// TwinCAT 3 PLC project SiasunDemo
// Title: ServoDriveDemo
// Company: Siasun
// ProjectVersion: 0.1.0
// ProgramVersion: 3.1.0.9
// libraries:
//   Tc2_EtherCAT, * (Beckhoff Automation GmbH)
//   Tc2_MC2, * (Beckhoff Automation GmbH)
//   Tc2_Standard, * (Beckhoff Automation GmbH)
//   Tc2_System, * (Beckhoff Automation GmbH)
//   Tc2_Utilities, * (Beckhoff Automation GmbH)
//   Tc2_XmlDataSrv, * (Beckhoff Automation GmbH)
//   Tc3_JsonXml, * (Beckhoff Automation GmbH)
//   Tc3_Module, * (Beckhoff Automation GmbH)
//   VisuDialogs, * (System)
// project tree:
//   DUTs/ Para.TcDUT, Struct_AxisDrive.TcDUT (not stored), Struct_AxisXmlRW.TcDUT, Struct_EndDrive.TcDUT, Struct_MotionPara.TcDUT, Struct_PLCVersion.TcDUT (not stored), Struct_AxisInfo.TcDUT (not stored), Struct_AxisStatus.TcDUT (not stored), Struct_ServoAccessParameters.TcDUT (not stored), Struct_ObservedParameters.TcDUT
//   / GlobalTextList.TcGTLO, PlcTask.TcTTO (not stored), 视图管理器.TcVMO (not stored)
//   POUs/CoeSdoRW/ AmsNetID_TO_TAmsNetID.TcPOU (not stored), FB_SDO_READ.TcPOU (not stored), FB_SDO_WRITE.TcPOU (not stored)
//   POUs/ FB_AxisOperate.TcPOU, MAIN.TcPOU (not stored)
//   VISUs/ StatJoint.TcVIS (not stored), StatJoint_6Axis.TcVIS
// real-time tasks:
//   TASK PlcTask: cycle T#4ms, priority 20, ADS port 350
//   TASK VISU_TASK: cycle T#200000us, priority 30, ADS port 351
//   TASK PlcTask1: cycle T#1ms, priority 21, ADS port 352
// motion (NC):
//   TASK NC-Task 1 SAF: cycle T#4ms, priority 4, ADS port 501
//   TASK NC-Task 1 SVB: cycle T#4ms, priority 8, ADS port 511
//   AXIS Axis 1 (id 1)
//     PositionAreaControl: Enable=false
//     TargetPosControl: Enable=false
//     OtherSettings: AllowMotionCmdToSlave=true
//     encoder EncType=19
//       EncPara: ScaleFactorNumerator=0.000686645507813, EncMode=3, MaxCount=#xffffffff, ReferenceSystem=1
//         Inc: RefSyncInverse=false
//     drive DrvType=16
//       DrvPara: MaxCount=#xffffffff, DriveControlDWord=#x00020000
//         Analog: TorqueSetpointScale=10
//         TimeComp: TaskDelayCycles=1
//     controller CtrType=1
//       CtrPara: PriorControlFactor=1
//         PosDiffControl: Enable=false
//         Observer: BandWidth=20
//   AXIS Axis 2 (id 2)
//     PositionAreaControl: Enable=false
//     TargetPosControl: Enable=false
//     OtherSettings: AllowMotionCmdToSlave=true
//     encoder EncType=19
//       EncPara: ScaleFactorNumerator=0.000686645507813, EncMode=3, MaxCount=#xffffffff, ReferenceSystem=1
//         Inc: RefSyncInverse=false
//     drive DrvType=16
//       DrvPara: MaxCount=#xffffffff, DriveControlDWord=#x00020000
//         Analog: TorqueSetpointScale=10
//         TimeComp: TaskDelayCycles=1
//     controller CtrType=1
//       CtrPara: PriorControlFactor=1
//         PosDiffControl: Enable=false
//         Observer: BandWidth=20
//   AXIS Axis 3 (id 3)
//     PositionAreaControl: Enable=false
//     TargetPosControl: Enable=false
//     OtherSettings: AllowMotionCmdToSlave=true
//     encoder EncType=19
//       EncPara: ScaleFactorNumerator=0.000686645507813, EncMode=3, MaxCount=#xffffffff, ReferenceSystem=1
//         Inc: RefSyncInverse=false
//     drive DrvType=16
//       DrvPara: MaxCount=#xffffffff, DriveControlDWord=#x00020000
//         TimeComp: TaskDelayCycles=1
//     controller CtrType=1
//       CtrPara: PriorControlFactor=1
//         PosDiffControl: Enable=false
//         Observer: BandWidth=20
//   AXIS Axis 4 (id 4)
//     PositionAreaControl: Enable=false
//     TargetPosControl: Enable=false
//     OtherSettings: AllowMotionCmdToSlave=true
//     encoder EncType=19
//       EncPara: ScaleFactorNumerator=0.000686645507813, EncMode=3, MaxCount=#xffffffff, ReferenceSystem=1
//         Inc: RefSyncInverse=false
//     drive DrvType=16
//       DrvPara: MaxCount=#xffffffff, DriveControlDWord=#x00020000
//         TimeComp: TaskDelayCycles=1
//     controller CtrType=1
//       CtrPara: PriorControlFactor=1
//         PosDiffControl: Enable=false
//         Observer: BandWidth=20
//   AXIS Axis 5 (id 5)
//     PositionAreaControl: Enable=false
//     TargetPosControl: Enable=false
//     OtherSettings: AllowMotionCmdToSlave=true
//     encoder EncType=19
//       EncPara: ScaleFactorNumerator=0.000686645507813, EncMode=3, MaxCount=#xffffffff, ReferenceSystem=1
//         Inc: RefSyncInverse=false
//     drive DrvType=16
//       DrvPara: MaxCount=#xffffffff, DriveControlDWord=#x00020000
//         TimeComp: TaskDelayCycles=1
//     controller CtrType=1
//       CtrPara: PriorControlFactor=1
//         PosDiffControl: Enable=false
//         Observer: BandWidth=20
//   AXIS Axis 6 (id 6)
//     PositionAreaControl: Enable=false
//     TargetPosControl: Enable=false
//     OtherSettings: AllowMotionCmdToSlave=true
//     encoder EncType=19
//       EncPara: ScaleFactorNumerator=0.000686645507813, EncMode=3, MaxCount=#xffffffff, ReferenceSystem=1
//         Inc: RefSyncInverse=false
//     drive DrvType=16
//       DrvPara: MaxCount=#xffffffff, DriveControlDWord=#x00020000
//         TimeComp: TaskDelayCycles=1
//     controller CtrType=1
//       CtrPara: PriorControlFactor=1
//         PosDiffControl: Enable=false
//         Observer: BandWidth=20
//   AXIS Axis 7 (id 7)
//     PositionAreaControl: Enable=false
//     TargetPosControl: Enable=false
//     OtherSettings: AllowMotionCmdToSlave=true
//     encoder EncType=19
//       EncPara: ScaleFactorNumerator=0.000686645507813, MaxCount=#xffffffff
//         Inc: RefSyncInverse=false
//     drive DrvType=16
//       DrvPara: MaxCount=#xffffffff
//         TimeComp: TaskDelayCycles=1
//     controller CtrType=1
//       CtrPara: PriorControlFactor=1
//         PosDiffControl: Enable=false
//         Observer: BandWidth=20
// I/O:
//   DEVICE Device 3 (EtherCAT), AmsNetId 172.16.3.61.4.1
//     Term 8 (EK1200) [EK1200-5000 EtherCAT Power supply (2A E-Bus)]
//       Term 8 (EK1110) [EK1110 EtherCAT extension]
//     Drive 9 (SERVO_ECAT) [SERVO_ECAT]
//     Drive 10 (SERVO_ECAT) [SERVO_ECAT]
//     Drive 11 (SERVO_ECAT) [SERVO_ECAT] (disabled)
//     Drive 12 (SERVO_ECAT) [SERVO_ECAT]
//     Drive 13 (SERVO_ECAT) [SERVO_ECAT]
//     Drive 14 (SERVO_ECAT) [SERVO_ECAT]
//     Box 15 (ECAT_EndIO) [ECAT_EndIO]
// variable links:
//   NC-Task 1 SAF/Axes/Axis 1 <-> Device 3 (EtherCAT)/Drive 9 (SERVO_ECAT)
//     Drive/Inputs/In/nDataIn3[0] <-> Input mapping 0/TorqueActualValue1
//     Drive/Inputs/In/nState1 <-> Input mapping 0/StatusWord
//     Drive/Inputs/In/nState2 <-> Input mapping 0/StatusWord @bit 8
//     Drive/Inputs/In/nState4 @bit 1 <-> WcState/InputToggle
//     Drive/Inputs/In/nState4 <-> WcState/WcState
//     Drive/Inputs/In/nState5 <-> Input mapping 0/ModesOfOperationDisplay
//     Drive/Outputs/Out/nCtrl1 <-> Output mapping 0/ControlWord
//     Drive/Outputs/Out/nCtrl2 <-> Output mapping 0/ControlWord @bit 8
//     Drive/Outputs/Out/nDataOut1 <-> Output mapping 0/TargetPosition
//     Enc/Inputs/In/nDataIn1 <-> Input mapping 0/PositionActualValue
//     Enc/Inputs/In/nState4 @bit 1 <-> WcState/InputToggle
//     Enc/Inputs/In/nState4 <-> WcState/WcState
//   NC-Task 1 SAF/Axes/Axis 2 <-> Device 3 (EtherCAT)/Drive 10 (SERVO_ECAT)
//     Drive/Inputs/In/nDataIn3[0] <-> Input mapping 0/TorqueActualValue1
//     Drive/Inputs/In/nState1 <-> Input mapping 0/StatusWord
//     Drive/Inputs/In/nState2 <-> Input mapping 0/StatusWord @bit 8
//     Drive/Inputs/In/nState4 @bit 1 <-> WcState/InputToggle
//     Drive/Inputs/In/nState4 <-> WcState/WcState
//     Drive/Inputs/In/nState5 <-> Input mapping 0/ModesOfOperationDisplay
//     Drive/Outputs/Out/nCtrl1 <-> Output mapping 0/ControlWord
//     Drive/Outputs/Out/nCtrl2 <-> Output mapping 0/ControlWord @bit 8
//     Drive/Outputs/Out/nDataOut1 <-> Output mapping 0/TargetPosition
//     Enc/Inputs/In/nDataIn1 <-> Input mapping 0/PositionActualValue
//     Enc/Inputs/In/nState4 @bit 1 <-> WcState/InputToggle
//     Enc/Inputs/In/nState4 <-> WcState/WcState
//   NC-Task 1 SAF/Axes/Axis 3 <-> Device 3 (EtherCAT)/Drive 11 (SERVO_ECAT)
//     Drive/Inputs/In/nDataIn3[0] <-> Input mapping 0/TorqueActualValue1
//     Drive/Inputs/In/nState1 <-> Input mapping 0/StatusWord
//     Drive/Inputs/In/nState2 <-> Input mapping 0/StatusWord @bit 8
//     Drive/Inputs/In/nState4 @bit 1 <-> WcState/InputToggle
//     Drive/Inputs/In/nState4 <-> WcState/WcState
//     Drive/Inputs/In/nState5 <-> Input mapping 0/ModesOfOperationDisplay
//     Drive/Outputs/Out/nCtrl1 <-> Output mapping 0/ControlWord
//     Drive/Outputs/Out/nCtrl2 <-> Output mapping 0/ControlWord @bit 8
//     Drive/Outputs/Out/nDataOut1 <-> Output mapping 0/TargetPosition
//     Enc/Inputs/In/nDataIn1 <-> Input mapping 0/PositionActualValue
//     Enc/Inputs/In/nState4 @bit 1 <-> WcState/InputToggle
//     Enc/Inputs/In/nState4 <-> WcState/WcState
//   NC-Task 1 SAF/Axes/Axis 4 <-> Device 3 (EtherCAT)/Drive 12 (SERVO_ECAT)
//     Drive/Inputs/In/nDataIn3[0] <-> Input mapping 0/TorqueActualValue1
//     Drive/Inputs/In/nState1 <-> Input mapping 0/StatusWord
//     Drive/Inputs/In/nState2 <-> Input mapping 0/StatusWord @bit 8
//     Drive/Inputs/In/nState4 @bit 1 <-> WcState/InputToggle
//     Drive/Inputs/In/nState4 <-> WcState/WcState
//     Drive/Inputs/In/nState5 <-> Input mapping 0/ModesOfOperationDisplay
//     Drive/Outputs/Out/nCtrl1 <-> Output mapping 0/ControlWord
//     Drive/Outputs/Out/nCtrl2 <-> Output mapping 0/ControlWord @bit 8
//     Drive/Outputs/Out/nDataOut1 <-> Output mapping 0/TargetPosition
//     Enc/Inputs/In/nDataIn1 <-> Input mapping 0/PositionActualValue
//     Enc/Inputs/In/nState4 @bit 1 <-> WcState/InputToggle
//     Enc/Inputs/In/nState4 <-> WcState/WcState
//   NC-Task 1 SAF/Axes/Axis 5 <-> Device 3 (EtherCAT)/Drive 13 (SERVO_ECAT)
//     Drive/Inputs/In/nDataIn3[0] <-> Input mapping 0/TorqueActualValue1
//     Drive/Inputs/In/nState1 <-> Input mapping 0/StatusWord
//     Drive/Inputs/In/nState2 <-> Input mapping 0/StatusWord @bit 8
//     Drive/Inputs/In/nState4 @bit 1 <-> WcState/InputToggle
//     Drive/Inputs/In/nState4 <-> WcState/WcState
//     Drive/Inputs/In/nState5 <-> Input mapping 0/ModesOfOperationDisplay
//     Drive/Outputs/Out/nCtrl1 <-> Output mapping 0/ControlWord
//     Drive/Outputs/Out/nCtrl2 <-> Output mapping 0/ControlWord @bit 8
//     Drive/Outputs/Out/nDataOut1 <-> Output mapping 0/TargetPosition
//     Enc/Inputs/In/nDataIn1 <-> Input mapping 0/PositionActualValue
//     Enc/Inputs/In/nState4 @bit 1 <-> WcState/InputToggle
//     Enc/Inputs/In/nState4 <-> WcState/WcState
//   NC-Task 1 SAF/Axes/Axis 6 <-> Device 3 (EtherCAT)/Drive 14 (SERVO_ECAT)
//     Drive/Inputs/In/nDataIn3[0] <-> Input mapping 0/TorqueActualValue1
//     Drive/Inputs/In/nState1 <-> Input mapping 0/StatusWord
//     Drive/Inputs/In/nState2 <-> Input mapping 0/StatusWord @bit 8
//     Drive/Inputs/In/nState4 @bit 1 <-> WcState/InputToggle
//     Drive/Inputs/In/nState4 <-> WcState/WcState
//     Drive/Inputs/In/nState5 <-> Input mapping 0/ModesOfOperationDisplay
//     Drive/Outputs/Out/nCtrl1 <-> Output mapping 0/ControlWord
//     Drive/Outputs/Out/nCtrl2 <-> Output mapping 0/ControlWord @bit 8
//     Drive/Outputs/Out/nDataOut1 <-> Output mapping 0/TargetPosition
//     Enc/Inputs/In/nDataIn1 <-> Input mapping 0/PositionActualValue
//     Enc/Inputs/In/nState4 @bit 1 <-> WcState/InputToggle
//     Enc/Inputs/In/nState4 <-> WcState/WcState
//   SiasunDemo/SiasunDemo Instance <-> Device 3 (EtherCAT)/Box 15 (ECAT_EndIO)
//     PlcTask Inputs/MAIN.EndInfo.EC_State <-> InfoData/State
//     PlcTask Inputs/MAIN.EndInfo.WC_State <-> WcState/WcState
//     PlcTask Inputs/MAIN.EndInfo.nSlaveAddr <-> InfoData/AdsAddr/port
//     PlcTask Inputs/MAIN.EndInfo.sNetID <-> InfoData/AdsAddr/netId
//   SiasunDemo/SiasunDemo Instance <-> Device 3 (EtherCAT)/Drive 10 (SERVO_ECAT)
//     PlcTask Inputs/MAIN.AxisOp[1].AxisDrive.InfoData_StateJoint <-> InfoData/State
//     PlcTask Inputs/MAIN.AxisOp[1].AxisDrive.Joint_PositionActual <-> Input mapping 0/AuxiliaryPositionActualValue
//     PlcTask Inputs/MAIN.AxisOp[1].AxisDrive.Joint_VelocityActual <-> Input mapping 0/AuxiliaryVelocityActualValue
//     PlcTask Inputs/MAIN.AxisOp[1].AxisDrive.MoveMode <-> Input mapping 0/ModesOfOperationDisplay
//     PlcTask Inputs/MAIN.AxisOp[1].AxisDrive.ServoErrId <-> Input mapping 0/ErrorCode
//     PlcTask Inputs/MAIN.AxisOp[1].AxisDrive.StatusWord <-> Input mapping 0/StatusWord
//     PlcTask Inputs/MAIN.AxisOp[1].AxisDrive.TorqueValue <-> Input mapping 0/CurrentActualvalue
//     PlcTask Inputs/MAIN.AxisOp[1].AxisDrive.WC_State <-> WcState/WcState
//     PlcTask Inputs/MAIN.AxisOp[1].AxisDrive.nSlaveAddr <-> InfoData/AdsAddr/port
//     PlcTask Inputs/MAIN.AxisOp[1].AxisDrive.sNetID <-> InfoData/AdsAddr/netId
//     PlcTask Outputs/MAIN.AxisOp[1].AxisDrive.TargetMode <-> Output mapping 0/ModesOfOperation
//     PlcTask Outputs/MAIN.AxisOp[1].AxisDrive.TargetTorque <-> Output mapping 0/TargetTorque
//     PlcTask Outputs/MAIN.AxisOp[1].AxisDrive.TargetVelocity <-> Output mapping 0/TargetVelocity
//   SiasunDemo/SiasunDemo Instance <-> Device 3 (EtherCAT)/Drive 11 (SERVO_ECAT)
//     PlcTask Inputs/MAIN.AxisOp[2].AxisDrive.InfoData_StateJoint <-> InfoData/State
//     PlcTask Inputs/MAIN.AxisOp[2].AxisDrive.Joint_PositionActual <-> Input mapping 0/AuxiliaryPositionActualValue
//     PlcTask Inputs/MAIN.AxisOp[2].AxisDrive.Joint_VelocityActual <-> Input mapping 0/AuxiliaryVelocityActualValue
//     PlcTask Inputs/MAIN.AxisOp[2].AxisDrive.MoveMode <-> Input mapping 0/ModesOfOperationDisplay
//     PlcTask Inputs/MAIN.AxisOp[2].AxisDrive.ServoErrId <-> Input mapping 0/ErrorCode
//     PlcTask Inputs/MAIN.AxisOp[2].AxisDrive.StatusWord <-> Input mapping 0/StatusWord
//     PlcTask Inputs/MAIN.AxisOp[2].AxisDrive.TorqueValue <-> Input mapping 0/CurrentActualvalue
//     PlcTask Inputs/MAIN.AxisOp[2].AxisDrive.WC_State <-> WcState/WcState
//     PlcTask Inputs/MAIN.AxisOp[2].AxisDrive.nSlaveAddr <-> InfoData/AdsAddr/port
//     PlcTask Inputs/MAIN.AxisOp[2].AxisDrive.sNetID <-> InfoData/AdsAddr/netId
//     PlcTask Outputs/MAIN.AxisOp[2].AxisDrive.TargetMode <-> Output mapping 0/ModesOfOperation
//     PlcTask Outputs/MAIN.AxisOp[2].AxisDrive.TargetTorque <-> Output mapping 0/TargetTorque
//     PlcTask Outputs/MAIN.AxisOp[2].AxisDrive.TargetVelocity <-> Output mapping 0/TargetVelocity
//   SiasunDemo/SiasunDemo Instance <-> Device 3 (EtherCAT)/Drive 12 (SERVO_ECAT)
//     PlcTask Inputs/MAIN.AxisOp[3].AxisDrive.InfoData_StateJoint <-> InfoData/State
//     PlcTask Inputs/MAIN.AxisOp[3].AxisDrive.Joint_PositionActual <-> Input mapping 0/AuxiliaryPositionActualValue
//     PlcTask Inputs/MAIN.AxisOp[3].AxisDrive.Joint_VelocityActual <-> Input mapping 0/AuxiliaryVelocityActualValue
//     PlcTask Inputs/MAIN.AxisOp[3].AxisDrive.MoveMode <-> Input mapping 0/ModesOfOperationDisplay
//     PlcTask Inputs/MAIN.AxisOp[3].AxisDrive.ServoErrId <-> Input mapping 0/ErrorCode
//     PlcTask Inputs/MAIN.AxisOp[3].AxisDrive.StatusWord <-> Input mapping 0/StatusWord
//     PlcTask Inputs/MAIN.AxisOp[3].AxisDrive.TorqueValue <-> Input mapping 0/CurrentActualvalue
//     PlcTask Inputs/MAIN.AxisOp[3].AxisDrive.WC_State <-> WcState/WcState
//     PlcTask Inputs/MAIN.AxisOp[3].AxisDrive.nSlaveAddr <-> InfoData/AdsAddr/port
//     PlcTask Inputs/MAIN.AxisOp[3].AxisDrive.sNetID <-> InfoData/AdsAddr/netId
//     PlcTask Outputs/MAIN.AxisOp[3].AxisDrive.TargetMode <-> Output mapping 0/ModesOfOperation
//     PlcTask Outputs/MAIN.AxisOp[3].AxisDrive.TargetTorque <-> Output mapping 0/TargetTorque
//     PlcTask Outputs/MAIN.AxisOp[3].AxisDrive.TargetVelocity <-> Output mapping 0/TargetVelocity
//   SiasunDemo/SiasunDemo Instance <-> Device 3 (EtherCAT)/Drive 13 (SERVO_ECAT)
//     PlcTask Inputs/MAIN.AxisOp[4].AxisDrive.InfoData_StateJoint <-> InfoData/State
//     PlcTask Inputs/MAIN.AxisOp[4].AxisDrive.Joint_PositionActual <-> Input mapping 0/AuxiliaryPositionActualValue
//     PlcTask Inputs/MAIN.AxisOp[4].AxisDrive.Joint_VelocityActual <-> Input mapping 0/AuxiliaryVelocityActualValue
//     PlcTask Inputs/MAIN.AxisOp[4].AxisDrive.MoveMode <-> Input mapping 0/ModesOfOperationDisplay
//     PlcTask Inputs/MAIN.AxisOp[4].AxisDrive.ServoErrId <-> Input mapping 0/ErrorCode
//     PlcTask Inputs/MAIN.AxisOp[4].AxisDrive.StatusWord <-> Input mapping 0/StatusWord
//     PlcTask Inputs/MAIN.AxisOp[4].AxisDrive.TorqueValue <-> Input mapping 0/CurrentActualvalue
//     PlcTask Inputs/MAIN.AxisOp[4].AxisDrive.WC_State <-> WcState/WcState
//     PlcTask Inputs/MAIN.AxisOp[4].AxisDrive.nSlaveAddr <-> InfoData/AdsAddr/port
//     PlcTask Inputs/MAIN.AxisOp[4].AxisDrive.sNetID <-> InfoData/AdsAddr/netId
//     PlcTask Outputs/MAIN.AxisOp[4].AxisDrive.TargetMode <-> Output mapping 0/ModesOfOperation
//     PlcTask Outputs/MAIN.AxisOp[4].AxisDrive.TargetTorque <-> Output mapping 0/TargetTorque
//     PlcTask Outputs/MAIN.AxisOp[4].AxisDrive.TargetVelocity <-> Output mapping 0/TargetVelocity
//   SiasunDemo/SiasunDemo Instance <-> Device 3 (EtherCAT)/Drive 14 (SERVO_ECAT)
//     PlcTask Inputs/MAIN.AxisOp[5].AxisDrive.InfoData_StateJoint <-> InfoData/State
//     PlcTask Inputs/MAIN.AxisOp[5].AxisDrive.Joint_PositionActual <-> Input mapping 0/AuxiliaryPositionActualValue
//     PlcTask Inputs/MAIN.AxisOp[5].AxisDrive.Joint_VelocityActual <-> Input mapping 0/AuxiliaryVelocityActualValue
//     PlcTask Inputs/MAIN.AxisOp[5].AxisDrive.MoveMode <-> Input mapping 0/ModesOfOperationDisplay
//     PlcTask Inputs/MAIN.AxisOp[5].AxisDrive.ServoErrId <-> Input mapping 0/ErrorCode
//     PlcTask Inputs/MAIN.AxisOp[5].AxisDrive.StatusWord <-> Input mapping 0/StatusWord
//     PlcTask Inputs/MAIN.AxisOp[5].AxisDrive.TorqueValue <-> Input mapping 0/CurrentActualvalue
//     PlcTask Inputs/MAIN.AxisOp[5].AxisDrive.WC_State <-> WcState/WcState
//     PlcTask Inputs/MAIN.AxisOp[5].AxisDrive.nSlaveAddr <-> InfoData/AdsAddr/port
//     PlcTask Inputs/MAIN.AxisOp[5].AxisDrive.sNetID <-> InfoData/AdsAddr/netId
//     PlcTask Outputs/MAIN.AxisOp[5].AxisDrive.TargetMode <-> Output mapping 0/ModesOfOperation
//     PlcTask Outputs/MAIN.AxisOp[5].AxisDrive.TargetTorque <-> Output mapping 0/TargetTorque
//     PlcTask Outputs/MAIN.AxisOp[5].AxisDrive.TargetVelocity <-> Output mapping 0/TargetVelocity
//   SiasunDemo/SiasunDemo Instance <-> Device 3 (EtherCAT)/Drive 9 (SERVO_ECAT)
//     PlcTask Inputs/MAIN.AxisOp[0].AxisDrive.InfoData_StateJoint <-> InfoData/State
//     PlcTask Inputs/MAIN.AxisOp[0].AxisDrive.Joint_PositionActual <-> Input mapping 0/AuxiliaryPositionActualValue
//     PlcTask Inputs/MAIN.AxisOp[0].AxisDrive.Joint_VelocityActual <-> Input mapping 0/AuxiliaryVelocityActualValue
//     PlcTask Inputs/MAIN.AxisOp[0].AxisDrive.MoveMode <-> Input mapping 0/ModesOfOperationDisplay
//     PlcTask Inputs/MAIN.AxisOp[0].AxisDrive.ServoErrId <-> Input mapping 0/ErrorCode
//     PlcTask Inputs/MAIN.AxisOp[0].AxisDrive.StatusWord <-> Input mapping 0/StatusWord
//     PlcTask Inputs/MAIN.AxisOp[0].AxisDrive.TorqueValue <-> Input mapping 0/CurrentActualvalue
//     PlcTask Inputs/MAIN.AxisOp[0].AxisDrive.nSlaveAddr <-> InfoData/AdsAddr/port
//     PlcTask Inputs/MAIN.AxisOp[0].AxisDrive.sNetID <-> InfoData/AdsAddr/netId
//     PlcTask Outputs/MAIN.AxisOp[0].AxisDrive.TargetMode <-> Output mapping 0/ModesOfOperation
//     PlcTask Outputs/MAIN.AxisOp[0].AxisDrive.TargetTorque <-> Output mapping 0/TargetTorque
//     PlcTask Outputs/MAIN.AxisOp[0].AxisDrive.TargetVelocity <-> Output mapping 0/TargetVelocity
//   SiasunDemo/SiasunDemo Instance <-> NC-Task 1 SAF/Axes/Axis 1
//     PlcTask Inputs/MAIN.AxisOp[0].AxisRef.NcToPlc <-> Outputs/ToPlc
//     PlcTask Outputs/MAIN.AxisOp[0].AxisRef.PlcToNc <-> Inputs/FromPlc
//   SiasunDemo/SiasunDemo Instance <-> NC-Task 1 SAF/Axes/Axis 2
//     PlcTask Inputs/MAIN.AxisOp[1].AxisRef.NcToPlc <-> Outputs/ToPlc
//     PlcTask Outputs/MAIN.AxisOp[1].AxisRef.PlcToNc <-> Inputs/FromPlc
//   SiasunDemo/SiasunDemo Instance <-> NC-Task 1 SAF/Axes/Axis 3
//     PlcTask Inputs/MAIN.AxisOp[2].AxisRef.NcToPlc <-> Outputs/ToPlc
//     PlcTask Outputs/MAIN.AxisOp[2].AxisRef.PlcToNc <-> Inputs/FromPlc
//   SiasunDemo/SiasunDemo Instance <-> NC-Task 1 SAF/Axes/Axis 4
//     PlcTask Inputs/MAIN.AxisOp[3].AxisRef.NcToPlc <-> Outputs/ToPlc
//     PlcTask Outputs/MAIN.AxisOp[3].AxisRef.PlcToNc <-> Inputs/FromPlc
//   SiasunDemo/SiasunDemo Instance <-> NC-Task 1 SAF/Axes/Axis 5
//     PlcTask Inputs/MAIN.AxisOp[4].AxisRef.NcToPlc <-> Outputs/ToPlc
//     PlcTask Outputs/MAIN.AxisOp[4].AxisRef.PlcToNc <-> Inputs/FromPlc
//   SiasunDemo/SiasunDemo Instance <-> NC-Task 1 SAF/Axes/Axis 6
//     PlcTask Inputs/MAIN.AxisOp[5].AxisRef.NcToPlc <-> Outputs/ToPlc
//     PlcTask Outputs/MAIN.AxisOp[5].AxisRef.PlcToNc <-> Inputs/FromPlc

// ---- DUTs/Para.TcDUT
TYPE Para :
STRUCT
	Id				:	DINT	:= -1;
	Name			:	STRING	:= 'None';
	Value			:	REAL	:= -999;
	qFmt			:	DINT	:= -999;
END_STRUCT
END_TYPE

// ---- DUTs/Struct_AxisXmlRW.TcDUT
TYPE Struct_AxisXmlRW :
STRUCT
//  xml read 

//ServoConfig/Download/Upload/ReadServoVersion-EtherCat/SelfCheckMode
	Download_State								:	INT := 0;
	ServoParameters_temp						:	ARRAY[0..99] OF PARA;
	
	XmlRead										:	FB_XmlSrvRead;
	Read_State									:	UINT := 0;
	CRC_Cal										:	UDINT;
	CRC_Read									:	UDINT;
	FilePath									:	ARRAY[0..6] OF STRING := ['C:\SiasunRobot\ServoConfig\Axis1.xml',
																			  'C:\SiasunRobot\ServoConfig\Axis2.xml',
																			  'C:\SiasunRobot\ServoConfig\Axis3.xml',
																			  'C:\SiasunRobot\ServoConfig\Axis4.xml',
																			  'C:\SiasunRobot\ServoConfig\Axis5.xml',
																			  'C:\SiasunRobot\ServoConfig\Axis6.xml',
																			  'C:\SiasunRobot\ServoConfig\Axis7.xml'];
	Config_State								:	INT := 0;
	Config_Para									:	PARA;
END_STRUCT
END_TYPE

// ---- DUTs/Struct_EndDrive.TcDUT
TYPE Struct_EndDrive :
STRUCT
    WC_State 				AT %I* 	:    	BIT;            // 参数可用标志 监控上电状态 1为断电 0为供电       
	EC_State 	AT %I* 	:    	UINT;            //  slave op state                    
	
   // systerm bar
	sNetID				AT %I*	:  	 	AmsNetID;
	nSlaveAddr			AT %I*	:  	 	UINT;
END_STRUCT
END_TYPE

// ---- DUTs/Struct_MotionPara.TcDUT
TYPE Struct_MotionPara :
STRUCT
	TargetPosition						:	LREAL;
	TargetPosition1						:	LREAL;
	TargetPosition2						:	LREAL;
	ReverseMotion_Velocity				:	LREAL	;
	AbsMotion_Velocity					:	LREAL	;
	TargetVelocity						:	LREAL	:=40;
	TargetAcceleration					:	LREAL	:=200;
	TargetDeceleration					:	LREAL	:=200;
	TargetJerk							:	LREAL	:=2000;
	TargetDistance						:	LREAL;
	StopDeceleration					:	LREAL	:=2000;
	Targetorque							:	INT;
	Repetitive							:	BOOL;
END_STRUCT
END_TYPE

// ---- DUTs/Struct_ObservedParameters.TcDUT
TYPE Struct_ObservedParameters :
STRUCT
	ADC_Iu						:	PARA;
	ADC_Iv						:	PARA;
	ADC_Iw						:	PARA;
	ADC_Udc						:	PARA;
	ADC_Temp_Board				:	PARA;
	ADC_Temp_Air				:	PARA;
	ADC_Temp_Motor				:	PARA;
	ADC_Idc						:	PARA;
	JointID						:	PARA;
	AlgorithmVersion			:	PARA;
	PolePairNumber				:	PARA;
	MmPerPolePair				:	PARA;
	LinesPerMm					:	PARA;
	GainEndEnc					:	PARA;
	GainMotEnc					:	PARA;
	StatusRead					:	PARA;
	tIconstRMS					:	PARA;
	tImaxRMS					:	PARA;
END_STRUCT
END_TYPE

// ---- POUs/FB_AxisOperate.TcPOU
FUNCTION_BLOCK FB_AxisOperate
VAR_INPUT
	AxisControlMode				:	INT;  // 1:  pos control  2: torque control
END_VAR
VAR_OUTPUT
END_VAR
VAR
	AxisRef										:	AXIS_REF;
	//Enable
	FB_ExtGenEnable								:	MC_ExtSetPointGenEnable;
	FB_ExtGenDisable							:	MC_ExtSetPointGenDisable;
	EnableTimer									:	TON;
	// read or write xml para of servo
	AxisXml 									: 	Struct_AxisXmlRW;
	//PLC Version
	PLC_Version									:	Struct_PLCVersion;
	// Motion para
	AxisMotionPara  							:	Struct_MotionPara;
	// AxisInfo
	AxisInfo									:	Struct_AxisInfo;
	//AxisStatus
	AxisStatus									:	Struct_AxisStatus;
	// Axis DRive
	AxisDrive									:	Struct_AxisDrive;
	//SDO R/W
	SDO_READ									:	FB_SDO_READ;
	SDO_WRITE									:	FB_SDO_WRITE;
	SDO_Buffer									:	DINT;
	//Parameters Design Local(relating to Parameter buffer list)
	ServoAccessParameters						:	Struct_ServoAccessParameters;
	ObservedParameters							:	Struct_observedParameters;
	count										:	INT;
	bServoParametersSet							:	BOOL:=FALSE;
	ServoParameters								:	ARRAY[0..99] OF PARA;
	//Error
	ServoError									:	BOOL;
	Error										:	BOOL;
	ErrId										:	DINT;
	NCErrorTrig									:	R_trig;
	EcComLoseTrig								:	F_trig;
	EcComLinkTrig								:	R_trig;
	// 
	Axis_num									:	INT;
	// Plc speed control
	AxisControlModeVar							:	INT;
	TargetCurrentOutput		 				    :   ARRAY [0..2] OF LREAL;
	Integral				  					:	ARRAY[0..3] OF  LREAL;	
	ErrOfSpeed									:	LREAL;

	test1 : LREAL:=0;
	test2 : LREAL:=0;
	test3 : LREAL:=0;
	
	(*傅里叶级数参数*)
	t 	  : LREAL;
	omega: LREAL := pi/15;
//TraPara: ARRAY[0..5, 0..6] OF LREAL:=[   0.0662 ,   -0.0642  ,  -0.1476  , 0.2446  ,  -0.1285 ,   -0.3109 ,  0.1071,
// 0.1153,    -0.0807,    -0.0397,   0.0184 , 0.1685  ,  -0.1337 ,   -0.0855,
// -0.1159,    0.0086,    0.0598,   -0.1741 ,   0.1077 ,   0.2901 ,  -0.0747,
// 0.2371,    -0.1044,    -0.0835,    -0.1411,   0.1452 ,   -0.0960 ,   -0.0620,
//  -0.2460,   0.0552,   0.0502,    -0.0016 ,   -0.0632 ,  0.2476 ,  0.0237,
//  -0.2545,   0.0170,   0.0093,   0.2473 ,   -0.0334 ,  0.0072 ,  0.0166];//实验轨迹,取优化后系数的负值，-x,除了轴3，轴三是正的
TraPara: ARRAY[0..5, 0..6] OF LREAL:=[   0.0015 ,   -0.0187  ,  0.0676  , -0.0357  ,  0.2127 ,   0.0342 ,  -0.1356,
0.0485,    -0.0121,    -0.0274,   0.1737 , -0.0235  ,  -0.2222 ,   0.0197,
-0.1282,    0.066,   0.0567,  0.0370 ,   -0.083 ,   0.0912 ,  0.0333,
0.0861,    -0.0603,    -0.066,    0.0863,   0.0435 ,   -0.1724 ,   -0.0089,
0.0084,   0.053,   0.1154,    0.0478 ,   0.0916 ,  -0.0562 ,  -0.0787,
0.0611,   -0.0845,   -0.1133,   0.0235 ,   0.0141 , -0.0846 ,  0.0188];//测试轨迹,全45度
 //TraPara: ARRAY[0..5, 0..6] OF LREAL:=[-0.0290 ,	0.0510 	,0.1741 ,	-0.1958, 	0.2306, 	0.2248 	,-0.1708 	,
//-0.1338 ,	-0.0993 ,	-0.1468 ,	-0.1535 ,	-0.0144, 	0.2873, 	0.0427 ,
//	0.0004 ,	0.1076 	,0.0151 	,-0.0004 ,	-0.3100 	,0.0000,	0.1708 ,
//	-0.1930 ,	0.0271, 	0.0701 ,	0.1017 ,	0.0718, 	0.0913 ,	-0.0569 ,
//	0.1965 ,	-0.0765 ,	-0.1024 ,	-0.1217 ,	0.0132 ,-0.0748 ,	0.0167 	,
//-0.2693 ,	0.0523 ,	0.0421, 	0.1500 ,	-0.0723, 	0.1193 	,0.0307 ];//全90度

	axis_move_reverse1						:	BOOL;
	axis_move_reverse2						: BOOL;
	move_reverse_lamp						: BOOL;
	EdgeTrigger 							: R_TRIG; // 上升沿检测
	
	

END_VAR

CASE AxisControlMode OF 
	0:
		IF AxisInfo.AxisStatus.NotMoving AND AxisInfo.AxisStatus.Ready AND AxisInfo.AxisStatus.Enabled THEN
			AxisControlModeVar := AxisControlMode;
		ELSE
			AxisControlModeVar := 0;
			Error := TRUE;
			ErrId := -2;
		END_IF
	1:		
			IF AxisDrive.TargetMode <> 8 THEN
				AxisDrive.TargetMode := 8;	
				AxisDrive.TargetTorque := 0;
				MC_ExtSetPointGenFeed(
					Position:=AxisInfo.ActualPosition, 
					Velocity:=1, 
					Acceleration:=1 , 
					Direction:=1 , 
					Axis:=AxisRef);			
			END_IF			
		
	2:
		IF AxisDrive.TargetMode <> 10 THEN
			AxisDrive.TargetMode := 10;
			AxisDrive.TargetTorque := AxisDrive.TorqueValue ;
		END_IF
			
END_CASE

METHOD Absolute_Motion : BOOL
VAR_INPUT
	axis_move_absolute						:	BOOL;
		Init_POS	:LREAL;
END_VAR
AxisDrive.MoveAbsolute( 
	Axis:=AxisRef , 
	Execute:=axis_move_absolute , 
	Position:= Init_POS+AxisMotionPara.TargetPosition , 
	Velocity:=AxisMotionPara.AbsMotion_Velocity , 
	Acceleration:=AxisMotionPara.TargetAcceleration , 
	Deceleration:=AxisMotionPara.TargetDeceleration , 
	Jerk:= AxisMotionPara.TargetJerk );

IF AxisDrive.MoveJog.Error THEN
	Error := TRUE;
	ErrId := AxisDrive.MoveAbsolute.ErrorID;
END_IF
END_METHOD

METHOD AxisConfig : BOOL
VAR_INPUT
	bExecute 							:	BOOL;
END_VAR
VAR
	pos									:	INT;
	temp								:	STRING;
END_VAR
(*					AxisConfig功能细则 Version20180831	
	功能描述:在关节上电后自动(被动强制过程, 否则伺服控制器无法正常工作)进行  参数配置
	使用方法:对成员函数AxisConfig进行调用
	实现细则: 
			 对单个关节实现上电后自动配置逻辑:
			 ->调用内部成员函数ReadServoVersion读取伺服驱动器软件与硬件版本号
			 ->等待标志位AxisStatus.SystemReady恢复FALSE
			 ->调用内部成员函数Read_Parameter读取本地对应关节配置参数列表至PLC本地Buffer
			 ->等待标志位AxisStatus.SystemReady恢复FALSE
			 ->调用内部成员函数Download_Parameter将参数列表下载至伺服驱动器
			 ->等待标志位AxisStatus.SystemReady恢复FALSE
			 ->进行上位机配置参数文件与伺服软件兼容性校验
			 ->若无任何报错并通过兼容性校验,AxisStatus.ConfigDone置True
		 	 PS: 其中各内部成员还是使用方法与实现细则请参考相关描述文件
	*)
IF NOT bExecute THEN
	AxisXml.Config_State := 0;
END_IF
CASE AxisXml.Config_State OF
	0://init
		AxisStatus.ConfigDone := FALSE;
		IF NOT AxisStatus.SystemReady THEN
			AxisStatus.SystemReady := TRUE;
		END_IF
		IF bExecute AND NOT Error THEN
			ServoParametersList();
			AxisXml.Config_State := 1;
		END_IF
	1://Read local file for current axis servo
		//IF NOT bServoParametersSet THEN
		Parameters_Read(TRUE);
		IF AxisStatus.SystemReady AND NOT Error THEN
			Parameters_Read(FALSE);
			AxisXml.Config_State := 2;
		END_IF
		//ELSE
		//	AxisXml.Config_State := 2;
		//END_IF
	2://Download Data to current axis servo
		Drive_Download(TRUE);
		IF AxisStatus.SystemReady AND NOT Error THEN
			Drive_Download(FALSE);
			AxisXml.Config_State := 3;
		END_IF	
	3://Axis Condig Done
		AxisStatus.ConfigDone:=TRUE;	//Current axis servo config done
END_CASE
END_METHOD

METHOD DataUpdate : BOOL
VAR_INPUT
	Axis_num_in							:	INT;
END_VAR
VAR
	i									:	UINT;
END_VAR
//Axis Motion Imformation
AxisInfo.Axis_OpMode := AxisDrive.MoveMode;
AxisInfo.PositionCmd := DINT_TO_LREAL(LREAL_TO_DINT(AxisRef.NcToPlc.SetPos*524288))/524288;//同步插值指令到实际指令count间的精度损失
AxisInfo.ActualPosition := AxisRef.NcToPlc.ActPos;
AxisInfo.ActualPositionCNT := AxisRef.NcToPlc.ActPos/0.000686645507813;
AxisInfo.ActualVelocity := AxisRef.NcToPlc.ActVelo;
AxisInfo.ActualAcceleration := AxisRef.NcToPlc.ActAcc;
AxisInfo.ActualTorque := AxisDrive.TorqueValue;
AxisInfo.AxisInfoDataStateJoint :=   AxisDrive.InfoData_StateJoint;

//  Axis motion cmd
AxisInfo.VelocityCmd := AxisRef.NcToPlc.SetVelo;
AxisInfo.Axis_TargetMode :=  AxisDrive.TargetMode;
AxisInfo.TorqueCmd :=   AxisDrive.TargetTorque;
//AxisDrive.TargetVelocity := LREAL_TO_DINT(AxisInfo.VelocityCmd);

//PLC Version
AxisInfo.PLC_Version := PLC_Version;
//Axis Basic Parameter
AxisRef.ReadStatus();
NCErrorTrig(CLK:=AxisRef.Status.Error,Q=>);
IF NCErrorTrig.Q AND NOT Error THEN
	Error := TRUE;
	ErrId := AxisRef.Status.ErrorID;
END_IF
Axis_num := Axis_num_in;
AxisInfo.AxisNum := Axis_num;
IF AxisInfo.AxisInfoDataStateJoint = 8 THEN
	AxisInfo.Axis_EcComOp := TRUE;
ELSE
	AxisInfo.Axis_EcComOp := FALSE;
END_IF
//EtherCAT Communication Error 
EcComLinkTrig(CLK:=AxisInfo.Axis_EcComOp,Q=>);
IF EcComLinkTrig.Q THEN
	AxisConfig(TRUE);
	IF Error AND ErrId = -99 THEN
		Error := FALSE;
		ErrId := 0;
	END_IF
END_IF
EcComLoseTrig(CLK:=AxisInfo.Axis_EcComOp,Q=>);
IF EcComLoseTrig.Q THEN
	FOR i := 0 TO 99 BY 1 DO
		AxisXml.ServoParameters_temp[i].Value := -999;
	END_FOR
	AxisConfig(FALSE);
	Error := TRUE;
	ErrId := -99 ;  // lose communication
END_IF
//Axis Status
AxisStatus.NotMoving := AxisRef.Status.NotMoving ;
AxisStatus.Standstill := AxisStatus.ConfigDone AND AxisStatus.NotMoving AND AxisStatus.SystemReady;
AxisStatus.Hasjob := NOT AxisStatus.Standstill;
IF ((AxisDrive.StatusWord AND 16#FFF7) <> AxisDrive.StatusWord) AND (AxisDrive.ServoErrId = 0) THEN
	AxisStatus.Ready := FALSE;
ELSE
	AxisStatus.Ready := TRUE;
END_IF
AxisInfo.AxisStatus := AxisStatus;

//Servo Err
AxisInfo.ServoError := ServoError;
AxisInfo.Error := Error OR ServoError;
IF ((AxisDrive.StatusWord AND 16#FFF7) <> AxisDrive.StatusWord) AND (AxisDrive.ServoErrId <> 0) AND (ErrId <> -99) THEN		//self defined error
	ServoError := TRUE; 
	AxisInfo.ErrId := AxisDrive.ServoErrId;
	AxisInfo.ErrId_Hex := DWORD_TO_HEXSTR(UDINT_TO_DWORD(AxisDrive.ServoErrId),8,FALSE);
ELSE
	ServoError := FALSE;
	AxisInfo.ErrId := ErrId;
	AxisInfo.ErrId_Hex := DINT_TO_STRING(ErrId);
END_IF
END_METHOD

METHOD Drive_Download : BOOL
VAR_INPUT
	Download_Para								:	BOOL;
END_VAR
VAR
	i											:	INT;
END_VAR
(*			Download Parameter功能细则 Version20181015	
	功能描述:根据本地伺服配置参数文件中的参数列表进行参数下载, 保存至伺服驱动器
	使用方法:对成员函数Download Parameter成员函数进行调用, 将输入Download_Para置True开始进行配置参数下载,下载过程中AxisStatus.SystemReady标志位将至FALSE,直至完成参数下载后置TRUE.将输入Download_Para置FALSE会复位功能函数
	实现细则: 
			 对单个配置参数的下载逻辑: 
			 ->确认PLC本地参数列表Buffer中的参数ID
			 ->若参数ID为有效ID,则提取其对应元素, 包括参数原始值及有效位参数
			 ->通过SDO写操作发送Head Mailbox请求配置参数下载操作, 下发的4个字节Head Mailbox从低位到高位分别为(括号中内容为注释):1(cmd);参数ID号;1(默认取1);0x02(SDO写操作对应驱动器通信channel)
			 ->确认Head Mailbox写操作完成
			 ->通过SDO写操作发送第一包数据内容,下发的2个16位数据内容从低位到高位分别为:INT(ABS(value*2^q))
			  (数据内容乘以2的有效位次方后取绝对值并将结果强制转换为int型);1/0(value符号标志位,若为负则取1,否则取0)
			 ->确认第一包数据内容完成写操作
			 ->通过SDO写操作发送第二包数据内容, 下发的2个16位数据内容从低位到高位分别为:参数ID号;1(写操作cmd);
			 ->确认第二包数据内容写操作完成
			 ->Finish
			 完成参数配置逻辑:
			 ->对单个配置参数下载进行循环, 直至在确认PLC本地参数列表Buffer中的参数ID为无效ID为止
	*)
IF NOT Download_Para THEN
	AxisXml.Download_State := 0;
END_IF
CASE AxisXml.Download_State OF
0://init
	SDO_WRITE(bExecute:=FALSE);
	SDO_Buffer := 0;
	count:=0;
	IF Download_Para AND AxisStatus.SystemReady THEN
		AxisStatus.SystemReady := FALSE;
		AxisXml.Download_State:=10;	
	END_IF
10://check parameter id
	AxisXml.Config_Para.Id := ServoParameters[count].Id;
	IF AxisXml.Config_Para.Id <> -1 THEN
		AxisXml.Config_Para.Value := ServoParameters[count].Value;
		AxisXml.Config_Para.qFmt := ServoParameters[count].qFmt;
		IF AxisXml.Config_Para.Value <> AxisXml.ServoParameters_temp[count].Value THEN
			AxisXml.ServoParameters_temp[count].Value := AxisXml.Config_Para.Value;
			AxisXml.Download_State:=11;
		ELSE
			count := count + 1;
		END_IF
	ELSE
		AxisXml.Download_State:= 20;
	END_IF
11://Write Head Mailbox
	SDO_Buffer := SHL(16#02,24)+SHL(1,16)+SHL(99,8)+1;	
	SDO_WRITE(bExecute:= TRUE, sNetID:=AxisDrive.sNetID, nSlaveAddr:=AxisDrive.nSlaveAddr, Buffer:= SDO_Buffer);
	IF NOT SDO_WRITE.bBusy AND NOT SDO_WRITE.bError AND SDO_WRITE.bDone THEN
		SDO_WRITE(bExecute:=FALSE);
		AxisXml.Download_State := 12;
	END_IF
12://Write Buffer[4..7]
	IF AxisXml.Config_Para.Value < 0 THEN									//Buffer[6..7]=sign		Buffer[4..5]=value*2^qFmt
		SDO_Buffer := SHL(1,16)+REAL_TO_DINT(ABS(AxisXml.Config_Para.Value)*EXPT(2,AxisXml.Config_Para.qFmt));
	ELSE
		SDO_Buffer := SHL(0,16)+REAL_TO_DINT(ABS(AxisXml.Config_Para.Value)*EXPT(2,AxisXml.Config_Para.qFmt));
	END_IF
	SDO_WRITE(bExecute:= TRUE, sNetID:=AxisDrive.sNetID, nSlaveAddr:=AxisDrive.nSlaveAddr, Buffer:= SDO_Buffer);
	IF NOT SDO_WRITE.bBusy AND NOT SDO_WRITE.bError AND SDO_WRITE.bDone THEN
		SDO_WRITE(bExecute:=FALSE);
		AxisXml.Download_State := 13;
	END_IF
13://Write Buffer[8..11]
	SDO_Buffer := SHL(16#1,16)+ AxisXml.Config_Para.Id;						//Buffer[10]=WriteCmd		Buffer[8..9]=Id
	SDO_WRITE(bExecute:= TRUE, sNetID:=AxisDrive.sNetID, nSlaveAddr:=AxisDrive.nSlaveAddr, Buffer:= SDO_Buffer);
	IF NOT SDO_WRITE.bBusy AND NOT SDO_WRITE.bError AND SDO_WRITE.bDone THEN
		SDO_WRITE(bExecute:=FALSE);
		count := count + 1;
		AxisXml.Download_State := 10;
	END_IF
20://Set tFPGA_RequestParaFlag Parameter
	AxisXml.Config_Para.Id := ServoAccessParameters.RequestParaFlag.Id;
	AxisXml.Config_Para.Value := 1;
	FOR i := 0 TO 99 BY 1 DO
		IF ServoParameters[i].Id = AxisXml.Config_Para.Id THEN
			AxisXml.Config_Para.qFmt := ServoParameters[i].qFmt;
		END_IF
	END_FOR
	AxisXml.Download_State := 21;
21://Write Head Mailbox
	SDO_Buffer := SHL(16#02,24)+SHL(1,16)+SHL(99,8)+1;	
	SDO_WRITE(bExecute:= TRUE, sNetID:=AxisDrive.sNetID, nSlaveAddr:=AxisDrive.nSlaveAddr, Buffer:= SDO_Buffer);
	IF NOT SDO_WRITE.bBusy AND NOT SDO_WRITE.bError AND SDO_WRITE.bDone THEN
		SDO_WRITE(bExecute:=FALSE);
		AxisXml.Download_State := 22;
	END_IF
22://Write Buffer[4..7]		Buffer[6..7]=sign		Buffer[4..5]=value*2^qFmt
	SDO_Buffer := SHL(0,16)+REAL_TO_DINT(ABS(AxisXml.Config_Para.Value)*EXPT(2,AxisXml.Config_Para.qFmt));						
	SDO_WRITE(bExecute:= TRUE, sNetID:=AxisDrive.sNetID, nSlaveAddr:=AxisDrive.nSlaveAddr, Buffer:= SDO_Buffer);
	IF NOT SDO_WRITE.bBusy AND NOT SDO_WRITE.bError AND SDO_WRITE.bDone THEN
		SDO_WRITE(bExecute:=FALSE);
		AxisXml.Download_State := 23;
	END_IF
23://Write Buffer[8..11]
	SDO_Buffer := SHL(16#1,16)+AxisXml.Config_Para.Id;						//Buffer[10]=WriteCmd		Buffer[8..9]=Id
	SDO_WRITE(bExecute:= TRUE, sNetID:=AxisDrive.sNetID, nSlaveAddr:=AxisDrive.nSlaveAddr, Buffer:= SDO_Buffer);
	IF NOT SDO_WRITE.bBusy AND NOT SDO_WRITE.bError AND SDO_WRITE.bDone THEN
		SDO_WRITE(bExecute:=FALSE);
		AxisStatus.SystemReady := FALSE;
		AxisXml.Download_State := 99;
	END_IF
99://finish & error
	AxisStatus.SystemReady := TRUE;
END_CASE

IF SDO_WRITE.bError THEN
	AxisStatus.SystemReady := TRUE;
	Error := TRUE;
	ErrId := SDO_WRITE.nErrId;
	AxisXml.Download_State := 99;
END_IF
END_METHOD

METHOD Enable_PosMode : BOOL
VAR_INPUT
	go_enable						:	BOOL;
END_VAR
(*						Version20180828				
	功能描述: 实现机器人控制器与关节实现通信后的使能与松抱闸
	使用方法: 对成员函数Enable进行调用, 将输入go_enalbe置TRUE
			 及会进行关节上使能与松抱闸操作, 将go_enable置false则会弹
			 抱闸掉使能
	实现细则: 
			 上使能逻辑: 下发关节进入位置模式指令,此时关节控制权限仍归
			 			伺服控制器->通过controlword上使能->通过
						statusword确认上使能->PLC打开外部值发生器
			 			->伺服驱动器控制关节进行松抱闸位移并松开抱闸,
			 			同时PLC下发位置指令实时跟随关节实际位置,等待伺
			 			服完成松抱闸操作->伺服进入位置模式,PLC接管实时
			 			位置接口->PLC关闭外部值发生器
			 下使能逻辑: PLC减速->通过controlword下发掉使能控制字->伺
			 			服减速至0.				   	 				*)
IF NOT go_enable THEN
	AxisDrive.Enable_State := 0;
END_IF
CASE AxisDrive.Enable_State OF
0://init
	IF AxisDrive.MoveMode <> 0 THEN
		AxisDrive.TargetMode := 0;
	END_IF
	AxisDrive.Enable(Axis:=AxisRef,Enable:=FALSE);
	AxisStatus.Enabled := FALSE;
	IF go_enable THEN
		AxisDrive.Enable_State := 1;
	END_IF
1://Op mode set and enable axis
	IF AxisDrive.TargetMode <> 8 THEN
		AxisDrive.TargetMode := 8;
	END_IF	
	
	AxisDrive.Enable(
		Axis:= AxisRef, 
		Enable:= go_enable, 
		Enable_Positive:= TRUE, 
		Enable_Negative:= TRUE, 
		Override:= 100);
		
	IF AxisDrive.Enable.Error THEN
		Error := TRUE;
		ErrId := AxisDrive.Enable.ErrorID;
	ELSIF AxisDrive.Enable.Status THEN
		AxisDrive.Enable_State := 2;	
	END_IF	
2://Enable axis external setpoint generator
	FB_ExtGenEnable(
		Axis:= AxisRef, 
		Execute:= TRUE, 
		Position:= 100000, 
		PositionType:= 1);
	IF FB_ExtGenEnable.Done AND FB_ExtGenEnable.Enabled THEN
		FB_ExtGenEnable(Axis:=AxisRef,Execute:=FALSE);
		AxisDrive.Enable_State := 3;
	ELSIF FB_ExtGenEnable.Error THEN
		Error := TRUE;
		ErrId := FB_ExtGenEnable.ErrorID;
	END_IF
3://make plc pos cmd follow actual position	
	MC_ExtSetPointGenFeed(
		Position:=AxisInfo.ActualPosition, 
		Velocity:=1, 
		Acceleration:=1 , 
		Direction:=1 , 
		Axis:=AxisRef);
	IF AxisDrive.MoveMode = 8 THEN
		AxisDrive.Enable_State := 4;
	END_IF
4://Disable external sepoint generator
	FB_ExtGenDisable(
		Axis:= AxisRef, 
		Execute:= TRUE);
	IF NOT FB_ExtGenDisable.Enabled AND FB_ExtGenDisable.Done THEN
		FB_ExtGenDisable(Axis:=AxisRef,Execute:=FALSE);
		AxisDrive.Enable_State := 5;
	ELSIF FB_ExtGenDisable.Error THEN
		Error := TRUE;
		ErrId := FB_ExtGenDisable.ErrorID;
	END_IF
5://Delay 1S
	EnableTimer(IN:=TRUE,PT:=TIME#1S,Q=>,ET=>);
	IF EnableTimer.Q THEN
		EnableTimer(IN:=FALSE);
		AxisDrive.Enable_State := 99;
	END_IF
99://finish
	AxisStatus.Enabled := TRUE;
END_CASE
END_METHOD

PROPERTY GetAxisInfo : Struct_AxisInfo
GET
GetAxisInfo := AxisInfo;
END_GET
END_PROPERTY

METHOD Home : BOOL
VAR_INPUT
	axis_move_absolute						:	BOOL;
	Init_POS	:LREAL;
END_VAR
VAR_OUTPUT
	move_init_done						:	BOOL;//初始运动完成
END_VAR

AxisDrive.MoveAbsolute(
	Axis:= AxisRef, 
	Execute:= axis_move_absolute, 
	Position:= Init_POS, 
	Velocity:= 1, 
	Acceleration:= , 
	Deceleration:= , 
	Jerk:= , 
	BufferMode:= , 
	Options:= , 
	Done=> move_init_done, 
	Busy=> , 
	Active=> , 
	CommandAborted=> , 
	Error=> , 
	ErrorID=> );
END_METHOD

METHOD Jog : BOOL
VAR_INPUT
	axis_jog_foward						:	BOOL;
	axis_jog_backwards					:	BOOL;
END_VAR
AxisDrive.MoveJog(
	Axis:= AxisRef, 
	JogForward:= axis_jog_foward, 
	JogBackwards:= axis_jog_backwards, 
	Mode:= MC_JOGMODE_CONTINOUS, 
	Position:= , 
	Velocity:= AxisMotionPara.TargetVelocity, 
	Acceleration:= AxisMotionPara.TargetAcceleration, 
	Deceleration:= AxisMotionPara.TargetDeceleration, 
	Jerk:= AxisMotionPara.TargetJerk);
	
IF AxisDrive.MoveJog.Error THEN
	Error := TRUE;
	ErrId := AxisDrive.MoveJog.ErrorID;

END_IF
END_METHOD

METHOD NotMovingReset : BOOL
VAR_INPUT
END_VAR
IF AxisDrive.MoveMode = 8 THEN
	Jog(FALSE,FALSE);
	Stop(FALSE);
ELSIF AxisDrive.MoveMode = 10 THEN
	PLCCurrentControl(
			CurrentControlMoveEnable:= FALSE , 
			PLCcycleInput:= 4, 
			TargetToque:= 0);
END_IF
END_METHOD

METHOD Parameters_Read : BOOL//Read Axis Servo Parameter From Local File
VAR_INPUT
	Read_Para									:	BOOL;
END_VAR
VAR
	i											:	UINT;
END_VAR
(*				Read Parameter功能细则 Version20181015		
	功能描述:读取计算机本地保存的关节伺服驱动器配置参数文件
	使用方法:将关节配置参数的.txt文件保存在C:\SiasunRobot\servo_config文件夹内,并确保文件名为"Axis(关节序号).xml(如:Axis1.xml)",对成员函数Read_Parameter进行调用,将输入Read_Para置TRUE,开始读取过程,待标志位AxisStatus.SystemReady回归TRUE代表完成读取;将输入Read_Para置TRUEead_Para置FALSE复位功能函数.
	实现细则: 
			 配置参数文件读取逻辑:
			 ->通过dataentry/PLC_Version读取xml中上位机版本号信息,供兼容性判定用
			 ->通过dataentry/CRC读取xml中CRC校验码信息,供CRC校验用
			 ->通过dataentry/ServoParameters读取伺服配置参数列表,供驱动器下载用
			 ->计算读取到的配置参数列表所对应的CRC,并与读取到的CRC校验码进行比对,进行校验,若通过则读取完成,否则CRC校验错误
	*)
if not Read_Para then
	AxisXml.Read_State := 0;
END_IF
CASE AxisXml.Read_State OF
0://init
	AxisXml.XmlRead(bExecute:=FALSE);
	IF Read_Para AND AxisStatus.SystemReady THEN
		AxisXml.CRC_Cal := 0;
		AxisStatus.SystemReady := FALSE;
		AxisXml.Read_State := 10;
	END_IF
10://Read PLC Version
	AxisXml.XmlRead(
		pSymAddr:= ADR(PLC_Version), 
		cbSymSize:= SIZEOF(PLC_Version), 
		sFilePath:= AxisXml.FilePath[Axis_Num], 
		sXPath:= '/dataentry/PLC_Version', 
		bExecute:= TRUE);
	IF NOT AxisXml.XmlRead.bError AND NOT AxisXml.XmlRead.bBusy THEN
		AxisXml.XmlRead(bExecute:=FALSE);
		AxisXml.Read_State := 11;
	END_IF
11://Read CRC Code
	AxisXml.XmlRead(
		pSymAddr:= ADR(AxisXml.CRC_Read), 
		cbSymSize:= SIZEOF(AxisXml.CRC_Read), 
		sFilePath:= AxisXml.FilePath[Axis_Num], 
		sXPath:= '/dataentry/CRC', 
		bExecute:= TRUE);
	IF NOT AxisXml.XmlRead.bError AND NOT AxisXml.XmlRead.bBusy THEN
		AxisXml.XmlRead(bExecute:=FALSE);
		AxisXml.Read_State := 12;
	END_IF
12://Read Servo Parameters List
	AxisXml.XmlRead(
		pSymAddr:= ADR(ServoParameters), 
		cbSymSize:= SIZEOF(ServoParameters), 
		sFilePath:= AxisXml.FilePath[Axis_Num], 
		sXPath:= '/dataentry/ServoParameters', 
		bExecute:= TRUE);
	IF NOT AxisXml.XmlRead.bError AND NOT AxisXml.XmlRead.bBusy THEN
		AxisXml.XmlRead(bExecute:=FALSE);
		AxisXml.Read_State := 20;
	END_IF
20://CRC Verification
	//FOR i := 0 TO 99 BY 1 DO
	//	AxisXml.CRC_Cal := AxisXml.CRC_Cal + DINT_TO_UDINT(ServoParameters[i].Id + REAL_TO_DINT(ServoParameters[i].Value) + ServoParameters[i].qFmt);
	//END_FOR
	//AxisXml.CRC_Cal := AxisXml.CRC_Cal + PLC_Version.Servo_Compatibility_high + PLC_Version.Servo_Compatibility_low + PLC_Version.PLC_Function;
	//AxisXml.CRC_Cal := NOT(AxisXml.CRC_cal);
	//AxisXml.CRC_Cal := WORD_TO_UDINT(F_DATA_TO_CRC16_CCITT(ADR(AxisXml.CRC_Cal),SIZEOF(AxisXml.CRC_Cal),16#0000));
	//IF AxisXml.CRC_Read <> AxisXml.CRC_cal THEN
	//	Error := TRUE;
	//	ErrId := 20;
	//END_IF
	AxisXml.Read_state := 99;
99://finish
	AxisStatus.SystemReady := TRUE;
END_CASE
IF AxisXml.XmlRead.bError THEN
	AxisStatus.SystemReady := TRUE;
	Error := TRUE;
	ErrId := AxisXml.XmlRead.nErrId;
END_IF
END_METHOD

METHOD PLCCurrentControl : BOOL  
VAR_INPUT
	CurrentControlMoveEnable		:	BOOL;
	PLCcycleInput					:	UDINT; // ms
	TargetToque						:	INT;
END_VAR
VAR
	PLCcycleReal			:	LREAL;
	SpeedControloutput		:	LREAL;
	SpeedControloutputLIMIT	:	LREAL;
END_VAR
PLCcycleReal := UDINT_TO_LREAL(PLCcycleInput/1000);

IF CurrentControlMoveEnable THEN	
	// SafeSetting安全
	IF TargetToque > 2000 THEN
		TargetToque:= 2000;
	ELSIF TargetToque< -2000 THEN
		TargetToque:= -2000;
	END_IF	
	
	
	PLCSpeedControl(
		SpeedControlEnable:= TRUE, 
		PLCcycle:= PLCcycleReal, 
		TargetSpeed:= 0, 
		ActualVelocity:= AxisInfo.ActualVelocity, 
		ba:= 0.01, 
		ksa:= 0.0, 
		kisa:= 0, 
		OutputOfControl=> SpeedControloutput);
	
	SpeedControloutputLIMIT := LIMIT(-32768,SpeedControloutput,32767) ;
	test2 := SpeedControloutputLIMIT;
	AxisDrive.TargetTorque := TargetToque + LREAL_TO_INT(SpeedControloutputLIMIT); 
	
ELSE
	PLCSpeedControl(
		SpeedControlEnable:= FALSE, 
		PLCcycle:= PLCcycleReal, 
		TargetSpeed:= 0, 
		ActualVelocity:= AxisInfo.ActualVelocity, 
		ba:= 0.01, 
		ksa:= 0, 
		kisa:= 0, 
		OutputOfControl=> SpeedControloutput);
	TargetToque :=0;
	SpeedControloutputLIMIT := 0 ;
	SpeedControloutput :=0;
	AxisDrive.TargetTorque := 0;
END_IF


test1 := SpeedControloutput;
test3 := TargetToque;
END_METHOD

METHOD PLCSpeedControl : BOOL
VAR_INPUT
	SpeedControlEnable			:	BOOL;
	PLCcycle			        :	LREAL;
	TargetSpeed					:	LREAL;   // 低速端 速度  °/s 设定值
	ActualVelocity				:	LREAL;   // 低速端速度 反馈值
	ba							:	LREAL;
	ksa							:	LREAL;
	kisa						:	LREAL;
END_VAR
VAR_OUTPUT
	OutputOfControl			    :	LREAL;
END_VAR
IF SpeedControlEnable THEN
	//ActualVelocity:=LIMT()	
	ErrOfSpeed:=TargetSpeed-ActualVelocity;

	Integral[0]:=ErrOfSpeed*PLCcycle+Integral[1];
	
	Integral[1]:=LIMIT(-1000,Integral[0],1000);
	
	Integral[2]:=Integral[1]*PLCcycle+Integral[3];
	
	Integral[3]:=LIMIT(-1000,Integral[2],1000);
	
	TargetCurrentOutput[0]:=ba*ErrOfSpeed+ksa*Integral[1]+kisa*Integral[3];
	
	TargetCurrentOutput[1]:=0.8*TargetCurrentOutput[0]+0.2*TargetCurrentOutput[2];
	TargetCurrentOutput[2]:=TargetCurrentOutput[1];
	
	OutputOfControl:=LIMIT(-10,TargetCurrentOutput[1],10);
ELSE
	OutputOfControl:=0;
	Integral[0] := 0;
	Integral[1] := 0;
	Integral[2] := 0;
	Integral[3] := 0;
	TargetCurrentOutput[0] := 0;
	TargetCurrentOutput[1] := 0;
	TargetCurrentOutput[2] := 0;
END_IF
END_METHOD

METHOD Reset : BOOL
VAR_INPUT
	Axis_Reset						:	BOOL;
END_VAR
AxisDrive.AxisReset(
	Axis:= AxisRef, 
	Execute:= Axis_Reset, 
	Done=> , 
	Busy=> , 
	Error=> , 
	ErrorID=> );
	
IF AxisDrive.AxisReset.Error THEN
	Error := TRUE;
	ErrId := AxisDrive.AxisReset.ErrorID;
	AxisDrive.AxisReset(Axis:=AxisRef,Execute:=FALSE);
ELSIF AxisDrive.AxisReset.Done AND NOT AxisDrive.AxisReset.Busy THEN
	Error := FALSE;
	ErrId := 0;
END_IF
END_METHOD

METHOD Reversing_Sequence : BOOL
VAR_INPUT
		Reversing_Sequence_Switch:BOOL;
		Init_POS	:LREAL;	
END_VAR
move_reverse_lamp:=Reversing_Sequence_Switch;
EdgeTrigger(CLK :=  Reversing_Sequence_Switch);
IF EdgeTrigger.Q  THEN
	axis_move_reverse1:=TRUE;
END_IF

IF Reversing_Sequence_Switch THEN
	

IF AxisDrive.MoveAbsolute1.Done THEN
	axis_move_reverse1:=FALSE;
	axis_move_reverse2:=TRUE;
ELSIF AxisDrive.MoveAbsolute2.Done THEN
	axis_move_reverse1:=TRUE;
	axis_move_reverse2:=FALSE;
END_IF
	   
IF AxisDrive.MoveAbsolute2.Done THEN
	AxisMotionPara.ReverseMotion_Velocity:=AxisMotionPara.ReverseMotion_Velocity+0.1;
END_IF

IF AxisMotionPara.ReverseMotion_Velocity>=1.1 THEN
	axis_move_reverse1:=FALSE;
	axis_move_reverse2:=FALSE;
END_IF

AxisDrive.MoveAbsolute1(
	Axis:=AxisRef , 
	Execute:=axis_move_reverse1 , 
	Position:=Init_POS+AxisMotionPara.TargetPosition1 , 
	Velocity:=AxisMotionPara.ReverseMotion_Velocity , 
	Acceleration:=AxisMotionPara.TargetAcceleration , 
	Deceleration:=AxisMotionPara.TargetDeceleration , 
	Jerk:= AxisMotionPara.TargetJerk  );
	
AxisDrive.MoveAbsolute2(
	Axis:=AxisRef , 
	Execute:=axis_move_reverse2 , 
	Position:=Init_POS+AxisMotionPara.TargetPosition2 , 
	Velocity:=AxisMotionPara.ReverseMotion_Velocity , 
	Acceleration:=AxisMotionPara.TargetAcceleration , 
	Deceleration:=AxisMotionPara.TargetDeceleration , 
	Jerk:= AxisMotionPara.TargetJerk  );
END_IF
END_METHOD

METHOD PRIVATE ServoParametersList : BOOL
VAR_INPUT
END_VAR
//Servo Cmd
ServoAccessParameters.ServoMode.Id := 84;
ServoAccessParameters.IsLocalCmd.Id := 61;
ServoAccessParameters.ServoOn.Id := 0;
ServoAccessParameters.RequestParaFlag.Id := 2;
//Position Control
ServoAccessParameters.BandWidth_Vel.Id := 17;
ServoAccessParameters.BandWidth_Posi.Id := 18;
ServoAccessParameters.BandWidth_Posi_int.Id := 23;
ServoAccessParameters.Low_Pass_BW.Id := 50;
ServoAccessParameters.DriectionReverse.Id := 19;

//Observed Parameters
ObservedParameters.ADC_Iu.Id := 65;
ObservedParameters.ADC_Iv.Id := 72;
ObservedParameters.ADC_Iw.Id := 73;
ObservedParameters.ADC_Udc.Id := 74;
ObservedParameters.ADC_Temp_Board.Id := 77;
ObservedParameters.ADC_Temp_Air.Id := 69;
ObservedParameters.ADC_Temp_Motor.Id := 75;
ObservedParameters.ADC_Idc.Id := 76;
ObservedParameters.JointID.Id := 60;
ObservedParameters.AlgorithmVersion.Id := 78;
ObservedParameters.PolePairNumber.Id := 46;
ObservedParameters.MmPerPolePair.Id := 11;
ObservedParameters.LinesPerMm.Id := 33;
ObservedParameters.GainEndEnc.Id := 36;
ObservedParameters.GainMotEnc.Id := 37;
ObservedParameters.StatusRead.Id := 62;
ObservedParameters.tIconstRMS.Id := 4;
ObservedParameters.tImaxRMS.Id := 5;
//Self Defined
ServoAccessParameters.StatusRequest.Id := 63;
//Error Protection
ServoAccessParameters.Over_Speed.Id := 58;
ServoAccessParameters.Over_PE.Id := 59;
ServoAccessParameters.Under_Volt.Id := 55;
ServoAccessParameters.Over_Volt.Id := 56;
ServoAccessParameters.Over_Curr.Id := 57;
ServoAccessParameters.Over_CrossPulseErr.Id := 38;
//Fault Mask
ServoAccessParameters.FaultMask_Low.Id := 54;
ServoAccessParameters.FaultMask_High.Id := 41;
END_METHOD

PROPERTY SetMotionPara : Struct_MotionPara
GET
SetMotionPara := AxisMotionPara;
END_GET
SET
IF ABS(SetMotionPara.TargetPosition1) <= 720 AND ABS(SetMotionPara.TargetPosition2) <= 720 AND ABS(SetMotionPara.TargetDistance+AxisInfo.ActualPosition) <=360 THEN
	AxisMotionPara := SetMotionPara;
ELSE
	AxisMotionPara.TargetPosition1 := AxisInfo.ActualPosition;
	AxisMotionPara.TargetPosition2 := AxisInfo.ActualPosition;
	AxisMotionPara.TargetDistance := 0;
	Error := TRUE;	
	ErrId := 0;
END_IF
END_SET
END_PROPERTY

PROPERTY SetServoParametersList : ARRAY[0..99] OF PARA;
SET
ServoParameters:=SetServoParametersList;
bServoParametersSet:=TRUE;
END_SET
END_PROPERTY

METHOD Stop : BOOL
VAR_INPUT
	axis_stop								:	BOOL;
END_VAR

IF AxisDrive.MoveMode = 8 THEN
	AxisDrive.AxisHalt(
	Axis:= AxisRef, 
	Execute:= axis_stop, 
	Deceleration:= AxisMotionPara.StopDeceleration, 
	Jerk:= AxisMotionPara.TargetJerk);
	
	IF AxisDrive.AxisHalt.Error THEN
		Error := TRUE;
		ErrId := AxisDrive.AxisHalt.ErrorID;
	END_IF

ELSIF AxisDrive.MoveMode = 10 THEN 
	AxisDrive.TargetTorque := 0;
END_IF
END_METHOD

METHOD Trajectory_Motion : BOOL
VAR_INPUT
	gen_enable	:BOOL;
	jointNum		:INT;
	Init_POS	:LREAL;
END_VAR
VAR_OUTPUT
	Position_desire: ARRAY[0..5] OF LREAL;
END_VAR
IF gen_enable THEN
	AxisDrive.GenEnable:=TRUE;
	AxisDrive.GenDisable:=FALSE;
ELSIF NOT gen_enable THEN
	AxisDrive.GenEnable:=FALSE;
	AxisDrive.GenDisable:=TRUE;
END_IF
AxisDrive.AxisExtSetPointGenEnable(
	Axis:=AxisRef , 
	Execute:= AxisDrive.GenEnable, 
	Position:=100000 , 
	PositionType:= 1 );
AxisDrive.AxisExtSetPointGenDisable(
	Axis:=AxisRef , 
	Execute:=AxisDrive.GenDisable);
IF AxisDrive.AxisExtSetPointGenEnable.Error THEN
		Error := TRUE;
		ErrId := AxisDrive.AxisExtSetPointGenEnable.ErrorID;	
ELSIF AxisDrive.AxisExtSetPointGenDisable.Error THEN
		Error := TRUE;
		ErrId := AxisDrive.AxisExtSetPointGenDisable.ErrorID;	
END_IF	
IF  AxisDrive.AxisExtSetPointGenEnable.Enabled AND AxisDrive.Enable.Status THEN
			AxisDrive.timer:=AxisDrive.timer+0.004;
			t:=AxisDrive.timer;	
MC_ExtSetPointGenFeed(
		Position:= Init_POS+180/pi*(TraPara[jointNum,0]/omega*SIN(omega*t) -TraPara[jointNum,1]/omega*COS(omega*t) +TraPara[jointNum,2]+TraPara[jointNum,3]/(2*omega)*SIN(2*omega*t) -TraPara[jointNum,4]/(2*omega)*COS(2*omega*t) +TraPara[jointNum,2]+TraPara[jointNum,5]/(3*omega)*SIN(3*omega*t) -TraPara[jointNum,6]/(3*omega)*COS(3*omega*t) +TraPara[jointNum,2]),
		Velocity:= 180/pi*(TraPara[jointNum,0]*COS(omega*t) +TraPara[jointNum,1]*SIN(omega*t)+TraPara[jointNum,3]*COS(2*omega*t) +TraPara[jointNum,4]*SIN(2*omega*t)+TraPara[jointNum,5]*COS(3*omega*t) +TraPara[jointNum,6]*SIN(3*omega*t)),
		Acceleration:=180/pi*(-TraPara[jointNum,0]*omega*SIN(omega*t) +TraPara[jointNum,1]*omega*COS(omega*t) -TraPara[jointNum,3]*(2*omega)*SIN(2*omega*t) +TraPara[jointNum,4]*(2*omega)*COS(2*omega*t) -TraPara[jointNum,5]*(3*omega)*SIN(3*omega*t) +TraPara[jointNum,6]*(3*omega)*COS(3*omega*t)) ,
		Direction:=1 , 
		Axis:=AxisRef);	//循环六次jointNum
//MC_ExtSetPointGenFeed(
//		Position:= Init_POS+110+180/pi*0.2-COS(0.2*pi*t)*180/pi*0.2,
//		Velocity:= 0.2*pi*SIN(0.2*pi*t)*180/pi*0.2,
//		Acceleration:=-0.2*pi*0.2*pi*COS(0.2*pi*t)*180/pi*0.2,
//		Direction:=1 , 
//		Axis:=AxisRef);	//测试

		Position_desire[jointNum-1]:=Init_POS+180/pi*(TraPara[jointNum,0]/omega*SIN(omega*t) -TraPara[jointNum,1]/omega*COS(omega*t) +TraPara[jointNum,2]+TraPara[jointNum,3]/(2*omega)*SIN(2*omega*t) -TraPara[jointNum,4]/(2*omega)*COS(2*omega*t) +TraPara[jointNum,2]+TraPara[jointNum,5]/(3*omega)*SIN(3*omega*t) -TraPara[jointNum,6]/(3*omega)*COS(3*omega*t) +TraPara[jointNum,2]);

END_IF
END_METHOD

END_FUNCTION_BLOCK

// ---- GlobalTextList.TcGTLO
TEXTLIST GlobalTextList
  70 = ' current control'
  45 = ' JOG+'
  4 = ' °'
  6 = ' °/s'
  56 = '%.1f'
  1 = '%.3f'
  35 = '%d'
  53 = '%f'
  17 = '%s'
  57 = '=>'
  89 = 'AbsMove'
  353 = 'AbsMoveDone:'
  102 = 'Absolute Motion'
  246 = 'ALL AXIS'
  926 = 'Axis1'
  749 = 'Axis2'
  349 = 'Axis3'
  415 = 'Axis4'
  748 = 'Axis5'
  117 = 'Axis6'
  58 = 'Bias:'
  68 = 'change to current control'
  67 = 'change to pos control'
  31 = 'ClearError'
  65 = 'Current Control：'
  49 = 'Current Job'
  50 = 'Current Job State'
  38 = 'Current Job：'
  64 = 'Current Mode：'
  71 = 'Current:'
  66 = 'CurrentMode'
  77 = 'CurrentModeDone?:'
  76 = 'Error Code Hex：'
  47 = 'Error Code：'
  39 = 'Error：'
  43 = 'Ext:'
  483 = 'ExtSetPointGenEnable'
  402 = 'ExtSetPointGenEnable:'
  54 = 'Global Speed Big:'
  55 = 'Global Speed Small:'
  52 = 'Global Speed:'
  33 = 'Go'
  22 = 'GoHome'
  594 = 'home'
  48 = 'Init'
  36 = 'J0:'
  51 = 'J1:'
  78 = 'J2:'
  79 = 'J3:'
  80 = 'J4:'
  81 = 'J5:'
  44 = 'JOG-'
  23 = 'MarkHome'
  21 = 'MarkZero'
  46 = 'MOVE'
  29 = 'MoveAbsolute:'
  28 = 'MoveRelative:'
  30 = 'MoveSpeed:'
  61 = 'None State'
  69 = 'pos control'
  72 = 'pos control to '
  73 = 'pos control to Current Ctrl'
  74 = 'pos Ctrl to Current Ctrl'
  75 = 'pos Ctrl to Current Ctrl:'
  24 = 'Position：'
  599 = 'Positon/ °'
  423 = 'Positon/ °:'
  675 = 'Positon/( °/s)'
  509 = 'Positon/()'
  42 = 'Power:'
  60 = 'Read  All'
  63 = 'Read Bias'
  34 = 'Run'
  20 = 'ServerOFF'
  41 = 'ServerOff'
  19 = 'ServerON'
  40 = 'ServerOn'
  962 = 'ServerOn(ALL AXIS)'
  340 = 'Speed/ (°/s):'
  455 = 'Speed/s:'
  25 = 'Speed:'
  37 = 'Speed：'
  26 = 'State:'
  32 = 'Stop'
  954 = 'TargetPosition/°:'
  156 = 'TargetPosition/°：'
  249 = 'TargetPosition1/°:'
  183 = 'TargetPosition2/°:'
  27 = 'TargetPosition：'
  399 = 'TargetPositon/ °:'
  82 = 'TargetSpeed/ (°/s):'
  1011 = 'TargetVelocity/°/s:'
  460 = 'TargetVelocity/°:'
  390 = 'Time/s'
  123 = 'Time/s:'
  337 = 'Trajectory Motion'
  59 = 'Write All'
  62 = 'Write Bias'
  0 = '伺服使能'
  3 = '伺服断开'
  13 = '停止运动'
  12 = '匀速运动'
  10 = '回零点'
  2 = '当前位置：'
  16 = '当前状态：'
  5 = '当前速度：'
  9 = '标记零点'
  18 = '清除错误'
  7 = '目标位置：'
  8 = '目标速度：'
  14 = '相对位置：'
  942 = '组块'
  11 = '转到目标位置'
  15 = '转动相对位置'
END_TEXTLIST

// ---- VISUs/StatJoint_6Axis.TcVIS
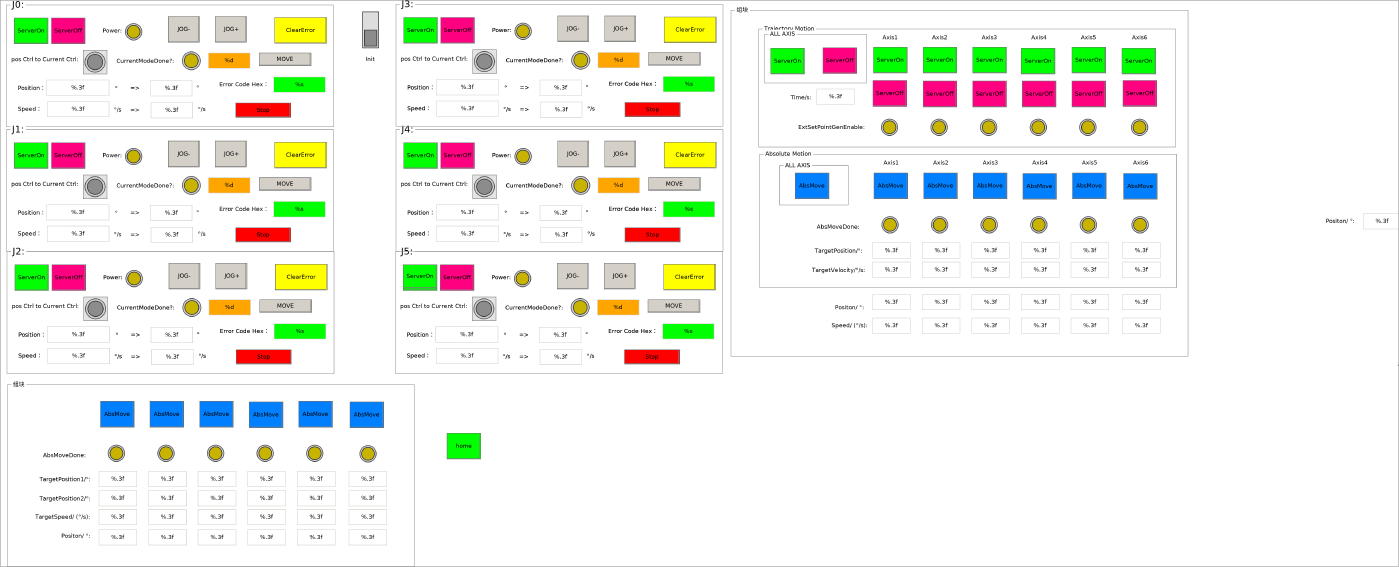
VISUALIZATION StatJoint_6Axis  // 2680x1087
    GroupBox (12,1 627x242), "J0:"
        Label (6,94 136x38), "pos Ctrl to Current Ctrl:"
        Label (13,192 64x32), "Speed："
        Label (224,191 45x38), "=>"
        Textfield (77,152 120x30), "%.3f", text variable: MAIN.AxisInfo[0].PositionCmd
        Label (198,154 22x29), "°"
        Textfield (78,193 119x30), "%.3f", text variable: MAIN.AxisMotionPara[0].TargetVelocity
            OnMouseClick: write the text variable via VisuDialogs.Numpad
        Label (193,195 37x29), "°/s"
        Button (86,33 65x50), "ServerOff", input disabled if: NOT MAIN.AxisOp[0].AxisInfo.AxisStatus.Ready
            toggle MAIN.HMI_AxisEnable[0]
        Button (514,32 100x50), "ClearError"
            tap MAIN.HMI_Axis_reset[0]
        Label (173,43 60x30), "Power:"
        Label (261,47 40x30)
        Button (310,30 60x50), "JOG-"
            tap MAIN.HMI_AxisJogBackwards[0]
        Button (400,30 60x50), "JOG+"
            tap MAIN.HMI_AxisJogFoward[0]
        Textfield (276,153 80x30), "%.3f", text variable: MAIN.AxisInfo[0].ActualPosition
        Label (354,153 22x29), "°"
        Label (354,194 37x29), "°/s"
        Textfield (277,195 80x30), "%.3f", text variable: MAIN.AxisInfo[0].ActualVelocity
        Textfield (387,100 80x30), "%d", text variable: MAIN.HMI_TargetTorque[0]
            OnMouseClick: write the text variable via VisuDialogs.Numpad
        Button (484,100 100x25), "MOVE"
            toggle MAIN.HMI_CurrentControlMove[0]
        Label (406,146 99x30), "Error Code Hex："
        Textfield (512,146 99x30), "%s", text variable: MAIN.AxisOp[0].AxisInfo.ErrId_Hex
        Label (224,149 45x38), "=>"
        Button (15,33 65x50), "ServerOn", input disabled if: NOT MAIN.AxisOp[0].AxisInfo.AxisStatus.Ready
            toggle MAIN.HMI_AxisEnable[0]
        PushSwitchLed (146,95 48x46), variable: MAIN.HMI_CurrentControlOfEnable[0], behaviour: TOGGLE, style: Switch-PushSwitchLed-Gray
        Label (18,149 62x38), "Position："
        Button (439,196 106x28), "Stop"
            tap MAIN.HMI_AxisStop[0]
        Lamp1 (225,40 38x40), variable: MAIN.AxisOp[0].AxisInfo.AxisStatus.Enabled, style: Lamp-Lamp1-Yellow
        Label (209,97 115x38), "CurrentModeDone?:"
        Lamp1 (334,94 41x43), variable: MAIN.HMI_AxisCurrentControlFlag[0], style: Lamp-Lamp1-Yellow
        Textfield (78,625 120x30), "%.3f", text variable: MAIN.AxisInfo[0].PositionCmd
        Label (199,627 22x29), "°"
        Label (14,665 64x32), "Speed："
        Textfield (79,666 119x30), "%.3f", text variable: MAIN.AxisMotionPara[0].TargetVelocity
            OnMouseClick: write the text variable via VisuDialogs.Numpad
        Label (194,668 37x29), "°/s"
        Button (87,506 65x50), "ServerOff", input disabled if: NOT MAIN.AxisOp[0].AxisInfo.AxisStatus.Ready
            toggle MAIN.HMI_AxisEnable[0]
        Button (515,505 100x50), "ClearError"
            tap MAIN.HMI_Axis_reset[0]
        Label (174,516 60x30), "Power:"
        Label (262,520 40x30)
        Button (311,503 60x50), "JOG-"
            tap MAIN.HMI_AxisJogBackwards[0]
        Button (401,503 60x50), "JOG+"
            tap MAIN.HMI_AxisJogFoward[0]
        Textfield (277,626 80x30), "%.3f", text variable: MAIN.AxisInfo[0].ActualPosition
        Label (355,626 22x29), "°"
        Label (355,667 37x29), "°/s"
        Textfield (278,668 80x30), "%.3f", text variable: MAIN.AxisInfo[0].ActualVelocity
        Textfield (388,573 80x30), "%d", text variable: MAIN.HMI_TargetTorque[0]
            OnMouseClick: write the text variable via VisuDialogs.Numpad
        Button (485,573 100x25), "MOVE"
            tap MAIN.HMI_CurrentControlMove[0]
        Label (407,619 99x30), "Error Code Hex："
        Textfield (513,619 99x30), "%s", text variable: MAIN.AxisOp[0].AxisInfo.ErrId_Hex
        Label (225,622 45x38), "=>"
        Label (225,664 45x38), "=>"
        Button (16,506 65x50), "ServerOn", input disabled if: NOT MAIN.AxisOp[0].AxisInfo.AxisStatus.Ready
            toggle MAIN.HMI_AxisEnable[0]
        PushSwitchLed (147,568 48x46), variable: MAIN.HMI_CurrentControlOfEnable[0], behaviour: TOGGLE, style: Switch-PushSwitchLed-Gray
        Label (19,622 62x38), "Position："
        Button (440,669 106x28), "Stop"
            tap MAIN.HMI_AxisStop[0]
        Lamp1 (226,513 38x40), variable: MAIN.AxisOp[0].AxisInfo.AxisStatus.Enabled, style: Lamp-Lamp1-Yellow
        Label (210,570 115x38), "CurrentModeDone?:"
        Lamp1 (335,567 41x43), variable: MAIN.HMI_AxisCurrentControlFlag[0], style: Lamp-Lamp1-Yellow
    DipSwitch (675,22 70x70), variable: MAIN.SiasunServoTestStart, behaviour: TOGGLE, style: Switch-DipSwitch-Gray
    Label (661,100 97x27), "Init"
    GroupBox (12,240 627x242), "J1:"
        Label (6,94 136x38), "pos Ctrl to Current Ctrl:"
        Textfield (77,152 120x30), "%.3f", text variable: MAIN.AxisInfo[1].PositionCmd
        Label (198,154 22x29), "°"
        Label (13,192 64x32), "Speed："
        Textfield (78,193 119x30), "%.3f", text variable: MAIN.AxisMotionPara[1].TargetVelocity
            OnMouseClick: write the text variable via VisuDialogs.Numpad
        Label (193,195 37x29), "°/s"
        Button (86,33 65x50), "ServerOff", input disabled if: NOT MAIN.AxisOp[1].AxisInfo.AxisStatus.Ready
            toggle MAIN.HMI_AxisEnable[1]
        Label (173,43 60x30), "Power:"
        Label (261,47 40x30)
        Button (310,30 60x50), "JOG-"
            tap MAIN.HMI_AxisJogBackwards[1]
        Button (400,30 60x50), "JOG+"
            tap MAIN.HMI_AxisJogFoward[1]
        Textfield (276,153 80x30), "%.3f", text variable: MAIN.AxisInfo[1].ActualPosition
        Label (354,153 22x29), "°"
        Label (354,194 37x29), "°/s"
        Textfield (277,195 80x30), "%.3f", text variable: MAIN.AxisInfo[1].ActualVelocity
        Textfield (387,100 80x30), "%d", text variable: MAIN.HMI_TargetTorque[1]
            OnMouseClick: write the text variable via VisuDialogs.Numpad
        Button (484,100 100x25), "MOVE"
            toggle MAIN.HMI_CurrentControlMove[1]
        Label (406,146 99x30), "Error Code Hex："
        Textfield (512,146 99x30), "%s", text variable: MAIN.AxisOp[1].AxisInfo.ErrId_Hex
        Label (224,149 45x38), "=>"
        Label (224,191 45x38), "=>"
        Button (15,33 65x50), "ServerOn", input disabled if: NOT MAIN.AxisOp[1].AxisInfo.AxisStatus.Ready
            toggle MAIN.HMI_AxisEnable[1]
        PushSwitchLed (146,95 48x46), variable: MAIN.HMI_CurrentControlOfEnable[1], behaviour: TOGGLE, style: Switch-PushSwitchLed-Gray
        Label (18,149 62x38), "Position："
        Button (439,196 106x28), "Stop"
            tap MAIN.HMI_AxisStop[1]
        Lamp1 (225,40 38x40), variable: MAIN.AxisOp[1].AxisInfo.AxisStatus.Enabled, style: Lamp-Lamp1-Yellow
        Label (209,97 115x38), "CurrentModeDone?:"
        Lamp1 (334,94 41x43), variable: MAIN.HMI_AxisCurrentControlFlag[1], style: Lamp-Lamp1-Yellow
        Button (514,32 100x50), "ClearError"
            tap MAIN.HMI_Axis_reset[1]
    GroupBox (13,474 627x242), "J2:"
        Label (6,94 136x38), "pos Ctrl to Current Ctrl:"
        Textfield (77,152 120x30), "%.3f", text variable: MAIN.AxisInfo[2].PositionCmd
        Label (198,154 22x29), "°"
        Label (13,192 64x32), "Speed："
        Textfield (78,193 119x30), "%.3f", text variable: MAIN.AxisMotionPara[2].TargetVelocity
            OnMouseClick: write the text variable via VisuDialogs.Numpad
        Label (193,195 37x29), "°/s"
        Button (86,33 65x50), "ServerOff", input disabled if: NOT MAIN.AxisOp[2].AxisInfo.AxisStatus.Ready
            toggle MAIN.HMI_AxisEnable[2]
        Button (514,32 100x50), "ClearError"
            tap MAIN.HMI_Axis_reset[2]
        Label (173,43 60x30), "Power:"
        Label (261,47 40x30)
        Button (310,30 60x50), "JOG-"
            tap MAIN.HMI_AxisJogBackwards[2]
        Button (400,30 60x50), "JOG+"
            tap MAIN.HMI_AxisJogFoward[2]
        Textfield (276,153 80x30), "%.3f", text variable: MAIN.AxisInfo[2].ActualPosition
        Label (354,153 22x29), "°"
        Label (354,194 37x29), "°/s"
        Textfield (277,195 80x30), "%.3f", text variable: MAIN.AxisInfo[2].ActualVelocity
        Textfield (387,100 80x30), "%d", text variable: MAIN.HMI_TargetTorque[2]
            OnMouseClick: write the text variable via VisuDialogs.Numpad
        Button (484,100 100x25), "MOVE"
            toggle MAIN.HMI_CurrentControlMove[2]
        Label (406,146 99x30), "Error Code Hex："
        Textfield (512,146 99x30), "%s", text variable: MAIN.AxisOp[2].AxisInfo.ErrId_Hex
        Label (224,149 45x38), "=>"
        Label (224,191 45x38), "=>"
        Button (15,33 65x50), "ServerOn", input disabled if: NOT MAIN.AxisOp[2].AxisInfo.AxisStatus.Ready
            toggle MAIN.HMI_AxisEnable[2]
        PushSwitchLed (146,95 48x46), variable: MAIN.HMI_CurrentControlOfEnable[2], behaviour: TOGGLE, style: Switch-PushSwitchLed-Gray
        Label (18,149 62x38), "Position："
        Button (439,196 106x28), "Stop"
            tap MAIN.HMI_AxisStop[2]
        Lamp1 (225,40 38x40), variable: MAIN.AxisOp[2].AxisInfo.AxisStatus.Enabled, style: Lamp-Lamp1-Yellow
        Label (209,97 115x38), "CurrentModeDone?:"
        Lamp1 (334,94 41x43), variable: MAIN.HMI_AxisCurrentControlFlag[2], style: Lamp-Lamp1-Yellow
        Textfield (821,152 120x30), "%.3f", text variable: MAIN.AxisInfo[0].PositionCmd
        Label (942,154 22x29), "°"
        Label (757,192 64x32), "Speed："
        Textfield (822,193 119x30), "%.3f", text variable: MAIN.AxisMotionPara[0].TargetVelocity
            OnMouseClick: write the text variable via VisuDialogs.Numpad
        Label (937,195 37x29), "°/s"
        Button (830,33 65x50), "ServerOff", input disabled if: NOT MAIN.AxisOp[0].AxisInfo.AxisStatus.Ready
            toggle MAIN.HMI_AxisEnable[0]
        Button (1258,32 100x50), "ClearError"
            tap MAIN.HMI_Axis_reset[0]
        Label (917,43 60x30), "Power:"
        Label (1005,47 40x30)
        Button (1054,30 60x50), "JOG-"
            tap MAIN.HMI_AxisJogBackwards[0]
        Button (1144,30 60x50), "JOG+"
            tap MAIN.HMI_AxisJogFoward[0]
        Textfield (1020,153 80x30), "%.3f", text variable: MAIN.AxisInfo[0].ActualPosition
        Label (1098,153 22x29), "°"
        Label (1098,194 37x29), "°/s"
        Textfield (1021,195 80x30), "%.3f", text variable: MAIN.AxisInfo[0].ActualVelocity
        Textfield (1131,100 80x30), "%d", text variable: MAIN.HMI_TargetTorque[0]
            OnMouseClick: write the text variable via VisuDialogs.Numpad
        Button (1228,100 100x25), "MOVE"
            tap MAIN.HMI_CurrentControlMove[0]
        Label (1150,146 99x30), "Error Code Hex："
        Textfield (1256,146 99x30), "%s", text variable: MAIN.AxisOp[0].AxisInfo.ErrId_Hex
        Label (968,149 45x38), "=>"
        Label (968,191 45x38), "=>"
        Button (759,33 65x50), "ServerOn", input disabled if: NOT MAIN.AxisOp[0].AxisInfo.AxisStatus.Ready
            toggle MAIN.HMI_AxisEnable[0]
        PushSwitchLed (890,95 48x46), variable: MAIN.HMI_CurrentControlOfEnable[0], behaviour: TOGGLE, style: Switch-PushSwitchLed-Gray
        Label (762,149 62x38), "Position："
        Button (1183,196 106x28), "Stop"
            tap MAIN.HMI_AxisStop[0]
        Lamp1 (969,40 38x40), variable: MAIN.AxisOp[0].AxisInfo.AxisStatus.Enabled, style: Lamp-Lamp1-Yellow
        Label (953,97 115x38), "CurrentModeDone?:"
        Lamp1 (1078,94 41x43), variable: MAIN.HMI_AxisCurrentControlFlag[0], style: Lamp-Lamp1-Yellow
    GroupBox (757,474 627x242), "J5:"
        Label (6,94 136x38), "pos Ctrl to Current Ctrl:"
        Textfield (77,152 120x30), "%.3f", text variable: MAIN.AxisInfo[5].PositionCmd
        Label (198,154 22x29), "°"
        Label (13,192 64x32), "Speed："
        Textfield (78,193 119x30), "%.3f", text variable: MAIN.AxisMotionPara[5].TargetVelocity
            OnMouseClick: write the text variable via VisuDialogs.Numpad
        Label (193,195 37x29), "°/s"
        Button (86,33 65x50), "ServerOff", input disabled if: NOT MAIN.AxisOp[5].AxisInfo.AxisStatus.Ready
            toggle MAIN.HMI_AxisEnable[5]
        Button (514,32 100x50), "ClearError"
            tap MAIN.HMI_Axis_reset[5]
        Label (173,43 60x30), "Power:"
        Label (261,47 40x30)
        Button (310,30 60x50), "JOG-"
            tap MAIN.HMI_AxisJogBackwards[5]
        Button (400,30 60x50), "JOG+"
            tap MAIN.HMI_AxisJogFoward[5]
        Textfield (276,153 80x30), "%.3f", text variable: MAIN.AxisInfo[5].ActualPosition
        Label (354,153 22x29), "°"
        Label (354,194 37x29), "°/s"
        Textfield (277,195 80x30), "%.3f", text variable: MAIN.AxisInfo[5].ActualVelocity
        Textfield (387,100 80x30), "%d", text variable: MAIN.HMI_TargetTorque[5]
            OnMouseClick: write the text variable via VisuDialogs.Numpad
        Button (484,100 100x25), "MOVE"
            toggle MAIN.HMI_CurrentControlMove[5]
        Label (406,146 99x30), "Error Code Hex："
        Textfield (512,146 99x30), "%s", text variable: MAIN.AxisOp[5].AxisInfo.ErrId_Hex
        Label (224,149 45x38), "=>"
        Label (224,191 45x38), "=>"
        Button (15,33 65x45), "ServerOn", input disabled if: NOT MAIN.AxisOp[5].AxisInfo.AxisStatus.Ready
            toggle MAIN.HMI_AxisEnable[5]
        PushSwitchLed (146,95 48x46), variable: MAIN.HMI_CurrentControlOfEnable[5], behaviour: TOGGLE, style: Switch-PushSwitchLed-Gray
        Label (18,149 62x38), "Position："
        Button (439,196 106x28), "Stop"
            tap MAIN.HMI_AxisStop[5]
        Lamp1 (225,40 38x40), variable: MAIN.AxisOp[5].AxisInfo.AxisStatus.Enabled, style: Lamp-Lamp1-Yellow
        Label (209,97 115x38), "CurrentModeDone?:"
        Lamp1 (334,94 41x43), variable: MAIN.HMI_AxisCurrentControlFlag[5], style: Lamp-Lamp1-Yellow
        Textfield (78,-82 120x30), "%.3f", text variable: MAIN.AxisInfo[0].PositionCmd
        Label (199,-80 22x29), "°"
        Label (14,-42 64x32), "Speed："
        Textfield (79,-41 119x30), "%.3f", text variable: MAIN.AxisMotionPara[0].TargetVelocity
            OnMouseClick: write the text variable via VisuDialogs.Numpad
        Label (194,-39 37x29), "°/s"
        Button (87,-201 65x50), "ServerOff", input disabled if: NOT MAIN.AxisOp[0].AxisInfo.AxisStatus.Ready
            toggle MAIN.HMI_AxisEnable[0]
        Button (515,-202 100x50), "ClearError"
            tap MAIN.HMI_Axis_reset[0]
        Label (174,-191 60x30), "Power:"
        Label (262,-187 40x30)
        Button (311,-204 60x50), "JOG-"
            tap MAIN.HMI_AxisJogBackwards[0]
        Button (401,-204 60x50), "JOG+"
            tap MAIN.HMI_AxisJogFoward[0]
        Textfield (277,-81 80x30), "%.3f", text variable: MAIN.AxisInfo[0].ActualPosition
        Label (355,-81 22x29), "°"
        Label (355,-40 37x29), "°/s"
        Textfield (278,-39 80x30), "%.3f", text variable: MAIN.AxisInfo[0].ActualVelocity
        Textfield (388,-134 80x30), "%d", text variable: MAIN.HMI_TargetTorque[0]
            OnMouseClick: write the text variable via VisuDialogs.Numpad
        Button (485,-134 100x25), "MOVE"
            tap MAIN.HMI_CurrentControlMove[0]
        Label (407,-88 99x30), "Error Code Hex："
        Textfield (513,-88 99x30), "%s", text variable: MAIN.AxisOp[0].AxisInfo.ErrId_Hex
        Label (225,-85 45x38), "=>"
        Label (225,-43 45x38), "=>"
        Button (16,-201 65x50), "ServerOn", input disabled if: NOT MAIN.AxisOp[0].AxisInfo.AxisStatus.Ready
            toggle MAIN.HMI_AxisEnable[0]
        PushSwitchLed (147,-139 48x46), variable: MAIN.HMI_CurrentControlOfEnable[0], behaviour: TOGGLE, style: Switch-PushSwitchLed-Gray
        Label (19,-85 62x38), "Position："
        Button (440,-38 106x28), "Stop"
            tap MAIN.HMI_AxisStop[0]
        Lamp1 (226,-194 38x40), variable: MAIN.AxisOp[0].AxisInfo.AxisStatus.Enabled, style: Lamp-Lamp1-Yellow
        Label (210,-137 115x38), "CurrentModeDone?:"
        Lamp1 (335,-140 41x43), variable: MAIN.HMI_AxisCurrentControlFlag[0], style: Lamp-Lamp1-Yellow
    GroupBox (758,240 627x242), "J4:"
        Label (6,94 136x38), "pos Ctrl to Current Ctrl:"
        Textfield (77,152 120x30), "%.3f", text variable: MAIN.AxisInfo[4].PositionCmd
        Label (198,154 22x29), "°"
        Label (13,192 64x32), "Speed："
        Textfield (78,193 119x30), "%.3f", text variable: MAIN.AxisMotionPara[4].TargetVelocity
            OnMouseClick: write the text variable via VisuDialogs.Numpad
        Label (193,195 37x29), "°/s"
        Button (86,33 65x50), "ServerOff", input disabled if: NOT MAIN.AxisOp[4].AxisInfo.AxisStatus.Ready
            toggle MAIN.HMI_AxisEnable[4]
        Button (514,32 100x50), "ClearError"
            tap MAIN.HMI_Axis_reset[4]
        Label (173,43 60x30), "Power:"
        Label (261,47 40x30)
        Button (310,30 60x50), "JOG-"
            tap MAIN.HMI_AxisJogBackwards[4]
        Button (400,30 60x50), "JOG+"
            tap MAIN.HMI_AxisJogFoward[4]
        Textfield (276,153 80x30), "%.3f", text variable: MAIN.AxisInfo[4].ActualPosition
        Label (354,153 22x29), "°"
        Label (354,194 37x29), "°/s"
        Textfield (277,195 80x30), "%.3f", text variable: MAIN.AxisInfo[4].ActualVelocity
        Textfield (387,100 80x30), "%d", text variable: MAIN.HMI_TargetTorque[4]
            OnMouseClick: write the text variable via VisuDialogs.Numpad
        Button (484,100 100x25), "MOVE"
            toggle MAIN.HMI_CurrentControlMove[4]
        Label (406,146 99x30), "Error Code Hex："
        Textfield (512,146 99x30), "%s", text variable: MAIN.AxisOp[4].AxisInfo.ErrId_Hex
        Label (224,149 45x38), "=>"
        Label (224,191 45x38), "=>"
        Button (15,33 65x50), "ServerOn", input disabled if: NOT MAIN.AxisOp[4].AxisInfo.AxisStatus.Ready
            toggle MAIN.HMI_AxisEnable[4]
        PushSwitchLed (146,95 48x46), variable: MAIN.HMI_CurrentControlOfEnable[4], behaviour: TOGGLE, style: Switch-PushSwitchLed-Gray
        Label (18,149 62x38), "Position："
        Button (439,196 106x28), "Stop"
            tap MAIN.HMI_AxisStop[4]
        Lamp1 (225,40 38x40), variable: MAIN.AxisOp[4].AxisInfo.AxisStatus.Enabled, style: Lamp-Lamp1-Yellow
        Label (209,97 115x38), "CurrentModeDone?:"
        Lamp1 (334,94 41x43), variable: MAIN.HMI_AxisCurrentControlFlag[4], style: Lamp-Lamp1-Yellow
        Group (13,-210 601x199)
            Textfield (64,122 120x30), "%.3f", text variable: MAIN.AxisInfo[0].PositionCmd
            Label (185,124 22x29), "°"
            Label (0,162 64x32), "Speed："
            Textfield (65,163 119x30), "%.3f", text variable: MAIN.AxisMotionPara[0].TargetVelocity
                OnMouseClick: write the text variable via VisuDialogs.Numpad
            Label (180,165 37x29), "°/s"
            Button (73,3 65x50), "ServerOff", input disabled if: NOT MAIN.AxisOp[0].AxisInfo.AxisStatus.Ready
                toggle MAIN.HMI_AxisEnable[0]
            Button (501,2 100x50), "ClearError"
                tap MAIN.HMI_Axis_reset[0]
            Label (160,13 60x30), "Power:"
            Label (248,17 40x30)
            Button (297,0 60x50), "JOG-"
                tap MAIN.HMI_AxisJogBackwards[0]
            Button (387,0 60x50), "JOG+"
                tap MAIN.HMI_AxisJogFoward[0]
            Textfield (263,123 80x30), "%.3f", text variable: MAIN.AxisInfo[0].ActualPosition
            Label (341,123 22x29), "°"
            Label (341,164 37x29), "°/s"
            Textfield (264,165 80x30), "%.3f", text variable: MAIN.AxisInfo[0].ActualVelocity
            Textfield (374,70 80x30), "%d", text variable: MAIN.HMI_TargetTorque[0]
                OnMouseClick: write the text variable via VisuDialogs.Numpad
            Button (471,70 100x25), "MOVE"
                tap MAIN.HMI_CurrentControlMove[0]
            Label (393,116 99x30), "Error Code Hex："
            Textfield (499,116 99x30), "%s", text variable: MAIN.AxisOp[0].AxisInfo.ErrId_Hex
            Label (211,119 45x38), "=>"
            Label (211,161 45x38), "=>"
            Button (2,3 65x50), "ServerOn", input disabled if: NOT MAIN.AxisOp[0].AxisInfo.AxisStatus.Ready
                toggle MAIN.HMI_AxisEnable[0]
            PushSwitchLed (133,65 48x46), variable: MAIN.HMI_CurrentControlOfEnable[0], behaviour: TOGGLE, style: Switch-PushSwitchLed-Gray
            Label (5,119 62x38), "Position："
            Button (426,166 106x28), "Stop"
                tap MAIN.HMI_AxisStop[0]
            Lamp1 (212,10 38x40), variable: MAIN.AxisOp[0].AxisInfo.AxisStatus.Enabled, style: Lamp-Lamp1-Yellow
            Label (196,67 115x38), "CurrentModeDone?:"
            Lamp1 (321,64 41x43), variable: MAIN.HMI_AxisCurrentControlFlag[0], style: Lamp-Lamp1-Yellow
    GroupBox (758,0 627x242), "J3:"
        Label (6,94 136x38), "pos Ctrl to Current Ctrl:"
        Textfield (77,152 120x30), "%.3f", text variable: MAIN.AxisInfo[3].PositionCmd
        Label (198,154 22x29), "°"
        Label (13,192 64x32), "Speed："
        Textfield (78,193 119x30), "%.3f", text variable: MAIN.AxisMotionPara[3].TargetVelocity
            OnMouseClick: write the text variable via VisuDialogs.Numpad
        Label (193,195 37x29), "°/s"
        Button (86,33 65x50), "ServerOff", input disabled if: NOT MAIN.AxisOp[3].AxisInfo.AxisStatus.Ready
            toggle MAIN.HMI_AxisEnable[3]
        Button (514,32 100x50), "ClearError"
            tap MAIN.HMI_Axis_reset[3]
        Label (173,43 60x30), "Power:"
        Label (261,47 40x30)
        Button (310,30 60x50), "JOG-"
            tap MAIN.HMI_AxisJogBackwards[3]
        Button (400,30 60x50), "JOG+"
            tap MAIN.HMI_AxisJogFoward[3]
        Textfield (276,153 80x30), "%.3f", text variable: MAIN.AxisInfo[3].ActualPosition
        Label (354,153 22x29), "°"
        Label (354,194 37x29), "°/s"
        Textfield (277,195 80x30), "%.3f", text variable: MAIN.AxisInfo[3].ActualVelocity
        Textfield (387,100 80x30), "%d", text variable: MAIN.HMI_TargetTorque[3]
            OnMouseClick: write the text variable via VisuDialogs.Numpad
        Button (484,100 100x25), "MOVE"
            toggle MAIN.HMI_CurrentControlMove[3]
        Label (406,146 99x30), "Error Code Hex："
        Textfield (512,146 99x30), "%s", text variable: MAIN.AxisOp[3].AxisInfo.ErrId_Hex
        Label (224,149 45x38), "=>"
        Label (224,191 45x38), "=>"
        Button (15,33 65x50), "ServerOn", input disabled if: NOT MAIN.AxisOp[3].AxisInfo.AxisStatus.Ready
            toggle MAIN.HMI_AxisEnable[3]
        PushSwitchLed (146,95 48x46), variable: MAIN.HMI_CurrentControlOfEnable[3], behaviour: TOGGLE, style: Switch-PushSwitchLed-Gray
        Label (18,149 62x38), "Position："
        Button (439,196 106x28), "Stop"
            tap MAIN.HMI_AxisStop[3]
        Lamp1 (225,40 38x40), variable: MAIN.AxisOp[3].AxisInfo.AxisStatus.Enabled, style: Lamp-Lamp1-Yellow
        Label (209,97 115x38), "CurrentModeDone?:"
        Lamp1 (334,94 41x43), variable: MAIN.HMI_AxisCurrentControlFlag[3], style: Lamp-Lamp1-Yellow
    Button (2678,700 2x0)
    GroupBox (1400,11 876x672), "组块"
        GroupBox (53,36 799x235), "Trajectory Motion"
            Button (220,43 65x50), "ServerOn"
                OnMouseClick: execute { Main.HMI_Tra_Motion[0]:=TRUE; }
            Button (219,107 65x50), "ServerOff"
                OnMouseClick: execute { Main.HMI_Tra_Motion[0]:=FALSE; }
            Lamp1 (232,177 38x40), variable: MAIN.AxisOp[0].AxisDrive.AxisExtSetPointGenEnable.Enabled, style: Lamp-Lamp1-Yellow
            Lamp1 (327,177 38x40), variable: MAIN.AxisOp[1].AxisDrive.AxisExtSetPointGenEnable.Enabled, style: Lamp-Lamp1-Yellow
            Lamp1 (422,177 38x40), variable: MAIN.AxisOp[2].AxisDrive.AxisExtSetPointGenEnable.Enabled, style: Lamp-Lamp1-Yellow
            Lamp1 (517,177 38x40), variable: MAIN.AxisOp[3].AxisDrive.AxisExtSetPointGenEnable.Enabled, style: Lamp-Lamp1-Yellow
            Lamp1 (612,177 38x40), variable: MAIN.AxisOp[4].AxisDrive.AxisExtSetPointGenEnable.Enabled, style: Lamp-Lamp1-Yellow
            Lamp1 (711,177 38x40), variable: MAIN.AxisOp[5].AxisDrive.AxisExtSetPointGenEnable.Enabled, style: Lamp-Lamp1-Yellow
            Button (315,43 65x50), "ServerOn"
                OnMouseClick: execute { Main.HMI_Tra_Motion[1]:=TRUE; }
            Button (410,43 65x50), "ServerOn"
                OnMouseClick: execute { Main.HMI_Tra_Motion[2]:=TRUE; }
            Button (600,43 65x50), "ServerOn"
                OnMouseClick: execute { Main.HMI_Tra_Motion[4]:=TRUE; }
            GroupBox (11,10 196x102), "ALL AXIS"
                Button (112,34 65x50), "ServerOff"
                    OnMouseClick: execute {
                        Main.HMI_Tra_Motion[0]:=FALSE;
                        Main.HMI_Tra_Motion[1]:=FALSE;
                        Main.HMI_Tra_Motion[2]:=FALSE;
                        Main.HMI_Tra_Motion[3]:=FALSE;
                        Main.HMI_Tra_Motion[4]:=FALSE;
                        Main.HMI_Tra_Motion[5]:=FALSE;
                    }
                Button (12,35 65x50), "ServerOn"
                    OnMouseClick: execute {
                        Main.HMI_Tra_Motion[0]:=TRUE;
                        Main.HMI_Tra_Motion[1]:=TRUE;
                        Main.HMI_Tra_Motion[2]:=TRUE;
                        Main.HMI_Tra_Motion[3]:=TRUE;
                        Main.HMI_Tra_Motion[4]:=TRUE;
                        Main.HMI_Tra_Motion[5]:=TRUE;
                    }
            Label (229,10 47x30), "Axis1"
            Label (324,10 47x30), "Axis2"
            Label (419,10 47x30), "Axis3"
            Label (514,10 47x30), "Axis4"
            Label (609,10 47x30), "Axis5"
            Label (707,10 47x30), "Axis6"
            Textfield (111,123 73x30), "%.3f", text variable: MAIN.AxisOp[0].AxisDrive.timer
            Label (58,125 47x30), "Time/s:"
            Label (72,182 136x30), "ExtSetPointGenEnable:"
            Button (315,108 65x50), "ServerOff"
                OnMouseClick: execute { Main.HMI_Tra_Motion[1]:=FALSE; }
            Button (410,108 65x50), "ServerOff"
                OnMouseClick: execute { Main.HMI_Tra_Motion[2]:=FALSE; }
            Button (505,108 65x50), "ServerOff"
                OnMouseClick: execute { Main.HMI_Tra_Motion[3]:=FALSE; }
            Button (600,108 65x50), "ServerOff"
                OnMouseClick: execute { Main.HMI_Tra_Motion[4]:=FALSE; }
            Button (698,107 65x50), "ServerOff"
                OnMouseClick: execute { Main.HMI_Tra_Motion[5]:=FALSE; }
            Button (503,45 65x50), "ServerOn"
                OnMouseClick: execute {  }
                OnMouseClick: execute { Main.HMI_Tra_Motion[3]:=TRUE; }
            Button (696,45 65x50), "ServerOn"
                OnMouseClick: execute { Main.HMI_Tra_Motion[5]:=TRUE; }
        GroupBox (55,276 799x264), "Absolute Motion"
            Label (229,10 47x30), "Axis1"
            Label (324,10 47x30), "Axis2"
            Label (419,10 47x30), "Axis3"
            Label (514,10 47x30), "Axis4"
            Label (609,10 47x30), "Axis5"
            Label (707,10 47x30), "Axis6"
            Textfield (1156,122 73x30), "%.3f", text variable: MAIN.AxisOP[0].AxisRef.NcToPlc.ActPos
            Textfield (1346,122 73x30), "%.3f", text variable: MAIN.AxisOP[2].AxisRef.NcToPlc.ActPos
            Textfield (1251,122 73x30), "%.3f", text variable: MAIN.AxisOP[1].AxisRef.NcToPlc.ActPos
            Textfield (1441,122 73x30), "%.3f", text variable: MAIN.AxisOP[3].AxisRef.NcToPlc.ActPos
            Textfield (1536,122 73x30), "%.3f", text variable: MAIN.AxisOP[4].AxisRef.NcToPlc.ActPos
            Textfield (1635,122 73x30), "%.3f", text variable: MAIN.AxisOP[5].AxisRef.NcToPlc.ActPos
            Label (1076,122 73x30), "Positon/ °:"
            GroupBox (38,22 132x84), "ALL AXIS"
                Button (30,22 65x50), "AbsMove"
                    OnMouseClick: execute {
                        Main.HMI_Abs_Motion[0]:=TRUE;
                        Main.HMI_Abs_Motion[1]:=TRUE;
                        Main.HMI_Abs_Motion[2]:=TRUE;
                        Main.HMI_Abs_Motion[3]:=TRUE;
                        Main.HMI_Abs_Motion[4]:=TRUE;
                        Main.HMI_Abs_Motion[5]:=TRUE;
                    }
            Button (219,44 65x50), "AbsMove"
                OnMouseClick: execute { main.HMI_Abs_Motion[0]:=TRUE; }
            Lamp1 (231,124 38x40), variable: MAIN.AxisOP[0].AxisDrive.MoveAbsolute.Active, style: Lamp-Lamp1-Yellow
            Lamp1 (326,124 38x40), variable: MAIN.AxisOP[1].AxisDrive.MoveAbsolute.Active, style: Lamp-Lamp1-Yellow
            Lamp1 (421,124 38x40), variable: MAIN.AxisOP[2].AxisDrive.MoveAbsolute.Active, style: Lamp-Lamp1-Yellow
            Lamp1 (516,124 38x40), variable: MAIN.AxisOP[3].AxisDrive.MoveAbsolute.Active, style: Lamp-Lamp1-Yellow
            Lamp1 (611,124 38x40), variable: MAIN.AxisOP[4].AxisDrive.MoveAbsolute.Active, style: Lamp-Lamp1-Yellow
            Lamp1 (710,124 38x40), variable: MAIN.AxisOP[5].AxisDrive.MoveAbsolute.Active, style: Lamp-Lamp1-Yellow
            Button (314,44 65x50), "AbsMove"
                OnMouseClick: execute { Main.HMI_Abs_Motion[1]:=TRUE; }
            Button (409,44 65x50), "AbsMove"
                OnMouseClick: execute { Main.HMI_Abs_Motion[2]:=TRUE; }
            Button (599,44 65x50), "AbsMove"
                OnMouseClick: execute { Main.HMI_Abs_Motion[4]:=TRUE; }
            Label (94,133 113x30), "AbsMoveDone:"
            Button (504,45 65x50), "AbsMove"
                OnMouseClick: execute {  }
                OnMouseClick: execute { Main.HMI_Abs_Motion[3]:=TRUE; }
            Button (697,45 65x50), "AbsMove"
                OnMouseClick: execute { Main.HMI_Abs_Motion[5]:=TRUE; }
            Textfield (216,178 73x30), "%.3f", text variable: MAIN.AxisOP[0].AxisMotionPara.TargetPosition
                OnMouseClick: write the text variable via VisuDialogs.Numpad
            Textfield (406,178 73x30), "%.3f", text variable: MAIN.AxisOP[2].AxisMotionPara.TargetPosition
                OnMouseClick: write the text variable via VisuDialogs.Numpad
            Textfield (311,178 73x30), "%.3f", text variable: MAIN.AxisOP[1].AxisMotionPara.TargetPosition
                OnMouseClick: write the text variable via VisuDialogs.Numpad
            Textfield (501,178 73x30), "%.3f", text variable: MAIN.AxisOP[3].AxisMotionPara.TargetPosition
                OnMouseClick: write the text variable via VisuDialogs.Numpad
            Textfield (596,178 73x30), "%.3f", text variable: MAIN.AxisOP[4].AxisMotionPara.TargetPosition
                OnMouseClick: write the text variable via VisuDialogs.Numpad
            Textfield (695,178 73x30), "%.3f", text variable: MAIN.AxisOP[5].AxisMotionPara.TargetPosition
                OnMouseClick: write the text variable via VisuDialogs.Numpad
            Label (95,179 113x30), "TargetPosition/°:"
            Textfield (216,215 73x30), "%.3f", text variable: MAIN.AxisOP[0].AxisMotionPara.AbsMotion_Velocity
                OnMouseClick: write the text variable via VisuDialogs.Numpad
        Textfield (271,553 73x30), "%.3f", text variable: MAIN.AxisOP[0].AxisRef.NcToPlc.ActPos
        Textfield (461,553 73x30), "%.3f", text variable: MAIN.AxisOP[2].AxisRef.NcToPlc.ActPos
        Textfield (366,553 73x30), "%.3f", text variable: MAIN.AxisOP[1].AxisRef.NcToPlc.ActPos
        Textfield (556,553 73x30), "%.3f", text variable: MAIN.AxisOP[3].AxisRef.NcToPlc.ActPos
        Textfield (651,553 73x30), "%.3f", text variable: MAIN.AxisOP[4].AxisRef.NcToPlc.ActPos
        Textfield (750,553 73x30), "%.3f", text variable: MAIN.AxisOP[5].AxisRef.NcToPlc.ActPos
        Textfield (271,598 73x30), "%.3f", text variable: MAIN.AxisOP[0].AxisRef.NcToPlc.ActVelo
        Label (191,553 73x51), "Positon/ °:"
        Label (191,598 73x30), "Speed/ (°/s):"
        Textfield (461,598 73x30), "%.3f", text variable: MAIN.AxisOP[2].AxisRef.NcToPlc.ActVelo
        Textfield (366,598 73x30), "%.3f", text variable: MAIN.AxisOP[1].AxisRef.NcToPlc.ActVelo
        Textfield (556,598 73x30), "%.3f", text variable: MAIN.AxisOP[3].AxisRef.NcToPlc.ActVelo
        Textfield (651,598 73x30), "%.3f", text variable: MAIN.AxisOP[4].AxisRef.NcToPlc.ActVelo
        Textfield (750,598 73x30), "%.3f", text variable: MAIN.AxisOP[5].AxisRef.NcToPlc.ActVelo
    Textfield (1861,502 73x30), "%.3f", text variable: MAIN.AxisOP[2].AxisMotionPara.AbsMotion_Velocity
        OnMouseClick: write the text variable via VisuDialogs.Numpad
    Textfield (1766,502 73x30), "%.3f", text variable: MAIN.AxisOP[1].AxisMotionPara.AbsMotion_Velocity
        OnMouseClick: write the text variable via VisuDialogs.Numpad
    Textfield (1956,502 73x30), "%.3f", text variable: MAIN.AxisOP[3].AxisMotionPara.AbsMotion_Velocity
        OnMouseClick: write the text variable via VisuDialogs.Numpad
    Textfield (2051,502 73x30), "%.3f", text variable: MAIN.AxisOP[4].AxisMotionPara.AbsMotion_Velocity
        OnMouseClick: write the text variable via VisuDialogs.Numpad
    Textfield (2150,502 73x30), "%.3f", text variable: MAIN.AxisOP[5].AxisMotionPara.AbsMotion_Velocity
        OnMouseClick: write the text variable via VisuDialogs.Numpad
    Label (1550,503 113x30), "TargetVelocity/°/s:"
    GroupBox (14,729 780x358), "组块"
        Button (178,40 65x50), "AbsMove"
            OnMouseClick: execute { main.HMI_Reverse_Motion[0]:=TRUE; }
        Lamp1 (190,120 38x40), variable: MAIN.AxisOP[0].move_reverse_lamp, style: Lamp-Lamp1-Yellow
        Lamp1 (285,120 38x40), variable: MAIN.AxisOP[1].move_reverse_lamp, style: Lamp-Lamp1-Yellow
        Lamp1 (380,120 38x40), variable: MAIN.AxisOP[2].move_reverse_lamp, style: Lamp-Lamp1-Yellow
        Lamp1 (475,120 38x40), variable: MAIN.AxisOP[3].move_reverse_lamp, style: Lamp-Lamp1-Yellow
        Button (273,40 65x50), "AbsMove"
            OnMouseClick: execute { main.HMI_Reverse_Motion[1]:=TRUE; }
        Button (368,40 65x50), "AbsMove"
            OnMouseClick: execute { Main.HMI_Reverse_Motion[2]:=TRUE; }
        Button (558,40 65x50), "AbsMove"
            OnMouseClick: execute { Main.HMI_Reverse_Motion[4]:=TRUE; }
        Label (53,129 113x30), "AbsMoveDone:"
        Button (463,41 65x50), "AbsMove"
            OnMouseClick: execute { Main.HMI_Reverse_Motion[3]:=TRUE; }
        Button (656,41 65x50), "AbsMove"
            OnMouseClick: execute { Main.HMI_Reverse_Motion[5]:=TRUE; }
        Textfield (175,174 73x30), "%.3f", text variable: MAIN.AxisOP[0].AxisMotionPara.TargetPosition1
            OnMouseClick: write the text variable via VisuDialogs.Numpad
        Textfield (365,174 73x30), "%.3f", text variable: MAIN.AxisOP[2].AxisMotionPara.TargetPosition1
            OnMouseClick: write the text variable via VisuDialogs.Numpad
        Textfield (270,174 73x30), "%.3f", text variable: MAIN.AxisOP[1].AxisMotionPara.TargetPosition1
            OnMouseClick: write the text variable via VisuDialogs.Numpad
        Textfield (460,174 73x30), "%.3f", text variable: MAIN.AxisOP[3].AxisMotionPara.TargetPosition1
            OnMouseClick: write the text variable via VisuDialogs.Numpad
        Textfield (555,174 73x30), "%.3f", text variable: MAIN.AxisOP[4].AxisMotionPara.TargetPosition1
            OnMouseClick: write the text variable via VisuDialogs.Numpad
        Textfield (654,174 73x30), "%.3f", text variable: MAIN.AxisOP[5].AxisMotionPara.TargetPosition1
            OnMouseClick: write the text variable via VisuDialogs.Numpad
        Label (54,175 113x30), "TargetPosition1/°:"
        Textfield (175,211 73x30), "%.3f", text variable: MAIN.AxisOP[0].AxisMotionPara.TargetPosition2
            OnMouseClick: write the text variable via VisuDialogs.Numpad
        Textfield (175,286 73x30), "%.3f", text variable: MAIN.AxisOP[0].AxisRef.NcToPlc.ActPos
        Textfield (365,286 73x30), "%.3f", text variable: MAIN.AxisOP[2].AxisRef.NcToPlc.ActPos
        Textfield (270,286 73x30), "%.3f", text variable: MAIN.AxisOP[1].AxisRef.NcToPlc.ActPos
        Textfield (460,286 73x30), "%.3f", text variable: MAIN.AxisOP[3].AxisRef.NcToPlc.ActPos
        Textfield (555,286 73x30), "%.3f", text variable: MAIN.AxisOP[4].AxisRef.NcToPlc.ActPos
        Textfield (654,286 73x30), "%.3f", text variable: MAIN.AxisOP[5].AxisRef.NcToPlc.ActPos
        Textfield (175,247 73x30), "%.3f", text variable: MAIN.AxisOP[0].AxisMotionPara.ReverseMotion_Velocity
            OnMouseClick: write the text variable via VisuDialogs.Numpad
        Label (95,273 73x51), "Positon/ °:"
        Label (44,247 124x30), "TargetSpeed/ (°/s):"
        Textfield (365,247 73x30), "%.3f", text variable: MAIN.AxisOP[2].AxisMotionPara.ReverseMotion_Velocity
            OnMouseClick: write the text variable via VisuDialogs.Numpad
        Textfield (270,247 73x30), "%.3f", text variable: MAIN.AxisOP[1].AxisMotionPara.ReverseMotion_Velocity
            OnMouseClick: write the text variable via VisuDialogs.NumpadExtended
        Textfield (460,247 73x30), "%.3f", text variable: MAIN.AxisOP[3].AxisMotionPara.ReverseMotion_Velocity
            OnMouseClick: write the text variable via VisuDialogs.Numpad
        Textfield (555,247 73x30), "%.3f", text variable: MAIN.AxisOP[4].AxisMotionPara.ReverseMotion_Velocity
            OnMouseClick: write the text variable via VisuDialogs.Numpad
        Textfield (654,247 73x30), "%.3f", text variable: MAIN.AxisOP[5].AxisMotionPara.ReverseMotion_Velocity
            OnMouseClick: write the text variable via VisuDialogs.Numpad
        Textfield (365,211 73x30), "%.3f", text variable: MAIN.AxisOP[2].AxisMotionPara.TargetPosition2
            OnMouseClick: write the text variable via VisuDialogs.Numpad
        Textfield (270,211 73x30), "%.3f", text variable: MAIN.AxisOP[1].AxisMotionPara.TargetPosition2
            OnMouseClick: write the text variable via VisuDialogs.Numpad
        Textfield (460,211 73x30), "%.3f", text variable: MAIN.AxisOP[3].AxisMotionPara.TargetPosition2
            OnMouseClick: write the text variable via VisuDialogs.Numpad
        Textfield (555,211 73x30), "%.3f", text variable: MAIN.AxisOP[4].AxisMotionPara.TargetPosition2
            OnMouseClick: write the text variable via VisuDialogs.Numpad
        Textfield (654,211 73x30), "%.3f", text variable: MAIN.AxisOP[5].AxisMotionPara.TargetPosition2
            OnMouseClick: write the text variable via VisuDialogs.Numpad
        Label (54,212 113x30), "TargetPosition2/°:"
        Lamp1 (570,120 38x40), variable: MAIN.AxisOP[4].move_reverse_lamp, style: Lamp-Lamp1-Yellow
        Lamp1 (672,121 38x40), variable: MAIN.AxisOP[5].move_reverse_lamp, style: Lamp-Lamp1-Yellow
    Button (856,830 65x50), "home"
        tap MAIN.home
END_VISUALIZATION
